// TIA Portal project "Projecto3Automação_1500_V18" (V18)

(* hardware
DEVICE "S71500/ET200MP station_1"  S7-1500 station
   slot 0: "Rail_0"  Rack  6ES7 590-1***0-0AA0
   slot 0: "PM 190W 120/230VAC"  PM 190W 120/230VAC  6EP1333-4BA00
   slot 1: "PLC_1"  CPU 1516-3 PN/DP  6ES7 516-3AN02-0AB0  V2.8
      slot 3: "CPU display_1"  6ES7591-1BA00-0AA0
      slot 32768: "PROFINET interface_1"  X1
         slot 32769: "Port_1"  X1 P1
         slot 32770: "Port_2"  X1 P2
      slot 33024: "PROFINET interface_2"  X2
         slot 33025: "Port_1"  X2 P1
      slot 33280: "DP interface_1"  X3
      slot 34817: "Virtual CP interface port_1"  Virtual CP interface port  Virtual CP interface port
   slot 2: "DI 32x24VDC HF_1"  DI 32x24VDC HF  6ES7 521-1BL00-0AB0  V2.2
   slot 3: "DQ 32x24VDC/0.5A HF_1"  DQ 32x24VDC/0.5A HF  6ES7 522-1BL01-0AB0  V1.1
   slot 4: "AI 8xU/I/RTD/TC ST_1"  AI 8xU/I/RTD/TC ST  6ES7 531-7KF00-0AB0  V2.2
   slot 5: "AQ 4xU/I ST_1"  AQ 4xU/I ST  6ES7 532-5HD00-0AB0  V2.2
DEVICE "PC station"  SIMATIC PC station
   slot 0: "PC station"  Rail  SIMATIC PC-Station  V1.0
      slot 125: "Stationmanager"  Station_Manager  V6.0.4
   slot 1: "HMI_RT_1"  WinCC RT Advanced  6AV2 104-0xxxx-xxxx  16.0.0.0
      slot 33792: "Computer interface"  Host interface
   slot 2: "IE general_1"  IE General  IE_CP  V8.2.0
DEVICE "S7-1500/ET200MP station_1"  S7-1500 station
   slot 0: "Rail_0"  Rack  6ES7 590-1***0-0AA0
   slot 1: "PLC_2"  CPU 1512C-1 PN  6ES7 512-1CK01-0AB0  V2.9
      slot 3: "CPU display_1"  6ES7591-1AA00-0AA0
      slot 32768: "PROFINET interface_1"  X1
         slot 32769: "Port_1"  X1 P1
         slot 32770: "Port_2"  X1 P2
      slot 34817: "Virtual CP interface port_1"  Virtual CP interface port  Virtual CP interface port
*)

// ===== PLC "PLC_1"  CPU 1516-3 PN/DP =====

VAR_GLOBAL   // PLC tag table "Default tag table"
   "Sensor Tapete 1 Entrada 1" AT %I10.0 : Bool;
   "Sensor Tapete 2 Entrada 2" AT %I10.1 : Bool;
   "Sensor Inicial Tapete 3 Saida 1" AT %I10.2 : Bool;
   "Sensor Final Tapete 3 Saida 1" AT %I10.3 : Bool;
   "Sensor Inicial Tapete 4 Saida 2" AT %I10.4 : Bool;
   "Sensor Final Tapete 4 Saida 2" AT %I10.5 : Bool;
   "Sensor Final Tapete 6 Saida 2" AT %I10.6 : Bool;
   "Sensor Final Tapete 7" AT %I10.7 : Bool;
   "Sensor  Grampo Aperto" AT %I11.0 : Bool;
   "Sensor Posicionador Cima/Baixo" AT %I11.1 : Bool;
   "Sensor Posicionador Frente/Tras" AT %I11.2 : Bool;
   "Sensor Posicionador Presença Peça" AT %I11.3 : Bool;
   "Sensor Saida Posto 1" AT %I11.4 : Bool;
   "Sensor Saida Posto 2" AT %I11.5 : Bool;
   "Sensor Saida Posto 3" AT %I11.6 : Bool;
   "Sensor Saida Posto 4" AT %I11.7 : Bool;
   "Sensor Saida Posto 5" AT %I12.0 : Bool;
   "Sensor Saida Posto 6" AT %I12.1 : Bool;
   "Emissor 1" AT %Q10.0 : Bool;
   "Tapete 1" AT %Q10.1 : Bool;
   "C. Maq. 1 Ativa" AT %Q10.2 : Bool;
   "C. Maq. 1 Parar" AT %Q10.3 : Bool;
   "C. Maq. 1 Bases/Tampas" AT %Q10.4 : Bool;
   "Emissor 2" AT %Q10.5 : Bool;
   "Tapete 2" AT %Q10.6 : Bool;
   "C. Maq. 2 Ativa" AT %Q10.7 : Bool;
   "C. Maq. 2 Parar" AT %Q11.0 : Bool;
   "C. Maq. 2 Bases/Tampas" AT %Q11.1 : Bool;
   "Grampo Aperto" AT %Q11.2 : Bool;
   "Grampo Levantar" AT %Q11.3 : Bool;
   "Posicionador Cima/Baixo" AT %Q11.4 : Bool;
   "Posicionador Frente/Tras" AT %Q11.5 : Bool;
   "Posicionador Vacuo" AT %Q11.6 : Bool;
   "Direcionador 1 Ligar" AT %Q12.0 : Bool;
   "Direcionador 1 Direita" AT %Q12.1 : Bool;
   "Direcionador 1 Esquerda" AT %Q12.2 : Bool;
   "Direcionador 2 Ligar" AT %Q12.3 : Bool;
   "Direcionador 2 Direita" AT %Q12.4 : Bool;
   "Direcionador 2 Esquerda" AT %Q12.5 : Bool;
   "Barreira Posto 3 e 5" AT %Q12.6 : Bool;
   "Barreira Posto 2 e 4" AT %Q12.7 : Bool;
   "C. Maq. 1 em Processo" AT %ID100 : DInt;
   "C. Maq. 2 em Processo" AT %ID104 : DInt;
   "Tapete 3" AT %QD100 : Real;
   "Tapete 4" AT %QD104 : Real;
   "Tapete 5" AT %QD108 : Real;
   "Tapete 6" AT %QD112 : Real;
   "Valvula Enchimento Tanque 1" AT %QD120 : Real;   // analog output manipulated value pump1
   "Valvula Descarga Tanque 1" AT %QD124 : Real;
   "Valvula Enchimento Tanque 2" AT %QD128 : Real;   // analog output manipulated value pump2
   "Valvula Descarga Tanque 2" AT %QD132 : Real;
   "Contador 1" AT %QD136 : DInt;
   "Contador 2" AT %QD140 : DInt;
   "Ordem de arranque" AT %M100.0 : Bool;
   "Ordem de paragem" AT %M100.1 : Bool;
   "M_Tapete1" AT %M103.0 : Bool;
   "M_Tapete2" AT %M103.1 : Bool;
   "M_Tapete3" AT %M103.2 : Bool;
   "M_Tapete4" AT %M103.3 : Bool;
   "M_Tapete5" AT %M103.4 : Bool;
   "M_Tapete6" AT %M103.5 : Bool;
   "M_Tapete7" AT %M103.6 : Bool;
   "V_Tapete3" AT %MD300 : Real;
   "V_Tapete4" AT %MD400 : Real;
   "V_Tapete5" AT %MD500 : Real;
   "V_Tapete6" AT %MD600 : Real;
   "V_Tapete7" AT %MD700 : Real;
   "Etapa_0" AT %M102.7 : Bool;
   "Etapa_1" AT %M103.7 : Bool;
   "Etapa_2" AT %M104.0 : Bool;
   "Etapa_3" AT %M104.1 : Bool;
   "Etapa_4" AT %M104.2 : Bool;
   "Etapa_5" AT %M104.3 : Bool;
   "Etapa_6" AT %M104.4 : Bool;
   "Etapa_7" AT %M104.5 : Bool;
   "Etapa_8" AT %M104.6 : Bool;
   "Etapa_9" AT %M104.7 : Bool;
   "Etapa_10" AT %M105.0 : Bool;
   "Etapa_11" AT %M105.1 : Bool;
   "Etapa_30" AT %M105.2 : Bool;
   "Etapa_31" AT %M105.3 : Bool;
   "Etapa_32" AT %M105.4 : Bool;
   "Etapa_33" AT %M105.5 : Bool;
   "Etapa_34" AT %M105.6 : Bool;
   "NPosto" AT %MW1000 : Int;
   "Etapa_12" AT %M105.7 : Bool;
   "Etapa_13" AT %M106.0 : Bool;
   "Etapa_14" AT %M106.1 : Bool;
   "Etapa_15" AT %M106.2 : Bool;
   "Etapa_20" AT %M106.3 : Bool;
   "Etapa_35" AT %M106.4 : Bool;
   "Etapa_36" AT %M106.5 : Bool;
   "Etapa_37" AT %M106.6 : Bool;
   "Etapa_38" AT %M106.7 : Bool;
   "Etapa_39" AT %M107.0 : Bool;
   "Etapa_40" AT %M107.1 : Bool;
   "Etapa_50" AT %M107.2 : Bool;
   "Empilhar" AT %M70.0 : Bool;
   "Sensor_Geral_Posto" AT %M170.0 : Bool;
   "Fim de ciclo" AT %M107.5 : Bool;
   "Sensor Grampo Levantar" AT %I12.2 : Bool;
   "Entrada_Base" AT %M107.6 : Bool;
   "Move Nposto 1" AT %M170.1 : Bool;
   "Etapa_100" AT %M150.0 : Bool;
   "Etapa_101" AT %M150.1 : Bool;
   "Etapa_102" AT %M150.2 : Bool;
   "Etapa_103" AT %M150.3 : Bool;
   "Etapa_104" AT %M150.4 : Bool;
   "Etapa_105" AT %M150.5 : Bool;
   "Etapa_106" AT %M150.6 : Bool;
   "Etapa_107" AT %M150.7 : Bool;
   "Etapa_110" AT %M151.0 : Bool;
   "Etapa_111" AT %M151.1 : Bool;
   "Etapa_112" AT %M151.2 : Bool;
   "Etapa_113" AT %M151.3 : Bool;
   "Etapa_114" AT %M151.4 : Bool;
   "Etapa_115" AT %M151.5 : Bool;
   "Etapa_116" AT %M151.6 : Bool;
   "Etapa_117" AT %M151.7 : Bool;
   "Etapa_120" AT %M152.0 : Bool;
   "Etapa_121" AT %M152.1 : Bool;
   "Etapa_122" AT %M152.2 : Bool;
   "Etapa_123" AT %M152.3 : Bool;
   "Etapa_124" AT %M152.4 : Bool;
   "Etapa_125" AT %M152.5 : Bool;
   "Etapa_126" AT %M152.6 : Bool;
   "Etapa_127" AT %M152.7 : Bool;
   "Etapa_130" AT %M153.0 : Bool;
   "Etapa_131" AT %M153.1 : Bool;
   "Etapa_132" AT %M153.2 : Bool;
   "Etapa_133" AT %M153.3 : Bool;
   "Etapa_134" AT %M153.4 : Bool;
   "Etapa_135" AT %M153.5 : Bool;
   "Etapa_136" AT %M153.6 : Bool;
   "Etapa_137" AT %M153.7 : Bool;
   "Etapa_150" AT %M155.0 : Bool;
   "Etapa_151" AT %M155.1 : Bool;
   "Etapa_152" AT %M155.2 : Bool;
   "Etapa_153" AT %M155.3 : Bool;
   "Etapa_154" AT %M155.4 : Bool;
   "Etapa_155" AT %M155.5 : Bool;
   "Etapa_156" AT %M155.6 : Bool;
   "Etapa_157" AT %M155.7 : Bool;
   "Pedido_Posic_Ao_Tapete_3" AT %M160.0 : Bool;
   "Pedido_Posic_Ao_Tapete_6" AT %M160.1 : Bool;
   "Pedido_Tap6_Ao_Tapete_4" AT %M160.2 : Bool;
   "Habilita_Remover_1" AT %M61.0 : Bool;
   "Habilita_Remover_2" AT %M61.1 : Bool;
   "Habilita_Remover_3" AT %M61.2 : Bool;
   "Habilita_Remover_4" AT %M61.3 : Bool;
   "Habilita_Remover_5" AT %M61.4 : Bool;
   "Habilita_Remover_6" AT %M61.5 : Bool;
   "Habilita_Máquina_1" AT %M61.6 : Bool;
   "Habilita_Máquina_2" AT %M61.7 : Bool;
   "Máquina1_Tampas" AT %M62.0 : Bool;
   "Máquina2_Tampas" AT %M62.1 : Bool;
   "Etapa_16" AT %M107.4 : Bool;
   "Scan_Estado_31" AT %M165.0 : Bool;
   "Contador_Remover_1" AT %MD10 : DWord;
   "Contador_Remover_2" AT %MD14 : DWord;
   "Contador_Remover_3" AT %MD18 : DWord;
   "Contador_Remover_4" AT %MD22 : DWord;
   "Contador_Remover_5" AT %MD26 : DWord;
   "Contador_Remover_6" AT %MD30 : DWord;
   "Start" AT %M100.2 : Bool;
   "Stop" AT %M100.3 : Bool;
   "Emergência" AT %M180.0 : Bool;
   "Reset" AT %M100.5 : Bool;
   "Nivel_Tanque_1" AT %ID108 : Real;   // analog Input actual level filing level Tank1
   "Nivel_Tanque_2" AT %ID112 : Real;   // analog Input actual level filing level Tank2
   "S1" AT %I150.0 : Bool;   // sudden setpoint change filing level 0 (0) or 700 (1)
   "Tapete 7" AT %QD116 : Real;
   "Algum_Remover_Habilitado" AT %M100.6 : Bool;
   "Algum_Máquina_Habilitada" AT %M100.7 : Bool;
   "Sem_Condições_Empilhar" AT %M101.0 : Bool;
   "Primeiro_Scan" AT %M200.0 : Bool;
   "Aviso_Sem_Condições_Empilhar" AT %M154.0 : Bool;
   "Aviso_Nenhuma_Máquina_Habilitada" AT %M158.0 : Bool;
   "Aviso_Nenhum_Remover_Habilitado" AT %M162.0 : Bool;
   "Contador_Remover_Total" AT %MD34 : DWord;
   "Aviso_Sem_Condições_Empilhar(1)" AT %MW154 : Int;
   "Aviso_Nenhuma_Máquina_Habilitada(1)" AT %MW158 : Int;
   "Aviso_Nenhum_Remover_Habilitado(1)" AT %MW162 : Int;
   "Contador_Máquina_1" AT %MD38 : DWord;
   "Contador_Máquina_2" AT %MD42 : DWord;
   "Nivel_1_convertido" AT %MD50 : Real;
   "Nivel_1_convertido_Scada" AT %ID60 : Real;
   "Reset Contadores Postos" AT %M700.0 : Bool;
   "Reset Contadores Maquinas" AT %M704.0 : Bool;
   "Nivel_2_convertido" AT %MD54 : Real;
   "Nivel_2_convertido_Scada" AT %ID64 : Real;
   "Emergencia Scada" AT %MW166 : Int;
   "Ret_value" AT %MW168 : Int;
   "Reset_Cont_Diario" AT %MD46 : DWord;
   "Tag_1" AT %MD174 : DWord;
   "Ordem de arranque s ordem paragem" AT %M100.4 : Bool;
   "Contador_Remover_1_Anterior" AT %MD310 : DWord;
   "Contador_Remover_2_Anterior" AT %MD314 : DWord;
   "Contador_Remover_3_Anterior" AT %MD318 : DWord;
   "Contador_Remover_4_Anterior" AT %MD322 : DWord;
   "Contador_Remover_5_Anterior" AT %MD326 : DWord;
   "Contador_Remover_6_Anterior" AT %MD330 : DWord;
   "Contador_Máquina_1_Anterior" AT %MD334 : DWord;
   "Contador_Máquina_2_Anterior" AT %MD338 : DWord;
   "Trigger_Contador" AT %M342.0 : Bool;
   "Set_vel_T3" AT %MD342 : Real;
   "Set_vel_T4" AT %MD346 : Real;
   "Set_vel_T5" AT %MD350 : Real;
   "Set_vel_T6" AT %MD354 : Real;
   "Set_vel_T7" AT %MD358 : Real;
   "Clock_1Hz" AT %M1100.5 : Bool;
   "Clock_2.5Hz" AT %M1100.2 : Bool;
   "Clock_2Hz" AT %M1100.3 : Bool;
END_VAR

DATA_BLOCK "Pulse"   // DB1
{ S7_Optimized_Access := 'TRUE' }
VERSION : 0.1
   VAR
      Pulse1 : Bool;
      Pulse2 : Bool;
      Pulse3 : Bool;
      Pulse4 : Bool;
      Pulse5 : Bool;
      Pulse6 : Bool;
      Pulse7 : Bool;
      Pulse8 : Bool;
      Pulse9 : Bool;
      Pulse10 : Bool;
      Pulse11 : Bool;
      Pulse12 : Bool;
      Pulse13 : Bool;
      Pulse14 : Bool;
      Pulse15 : Bool;
      Pulse16 : Bool;
      Pulse17 : Bool;
      Pulse18 : Bool;
      Pulse19 : Bool;
      Pulse20 : Bool;
      Pulse21 : Bool;
      Pulse22 : Bool;
      Pulse23 : Bool;
      Pulse24 : Bool;
      pulse25 : Bool;
      pulse26 : Bool;
      pulse27 : Bool;
      pulse28 : Bool;
      pulse29 : Bool;
      pulse30 : Bool;
      pulse31 : Bool;
      pulse32 : Bool;
      pulse33 : Bool;
   END_VAR
BEGIN
END_DATA_BLOCK

DATA_BLOCK "PLC1_Data_Sent"   // DB19
{ S7_Optimized_Access := 'FALSE' }
VERSION : 0.1
   VAR
      Contador_Remover_1 : DWord;
      Contador_Remover_2 : DWord;
      Contador_Remover_3 : DWord;
      Contador_Remover_4 : DWord;
      Contador_Remover_5 : DWord;
      Contador_Remover_6 : DWord;
      Contador_Remover_Total : DWord;
      Contador_Máquina_1 : DWord;
      Contador_Máquina_2 : DWord;
      "Valvula Enchimento Tanque 1" : Real;
      "Valvula Descarga Tanque 1" : Real;
      "Valvula Enchimento Tanque 2" : Real;
      "Valvula Descarga Tanque 2" : Real;
      Nivel_1_convertido_Scada : Real;
      Nivel_2_convertido_Scada : Real;
      Aviso_Nenhuma_Máquina_Habilitada : Bool;
      Aviso_Nenhum_Remover_Habilitado : Bool;
      Aviso_Sem_Condições_Empilhar : Bool;
      OUT_Set_vel_T3 : Real;
      OUT_Set_vel_T4 : Real;
      OUT_Set_vel_T5 : Real;
      OUT_Set_vel_T6 : Real;
      OUT_Set_vel_T7 : Real;
   END_VAR
BEGIN
END_DATA_BLOCK

DATA_BLOCK "PLC1_Data_Received"   // DB22
{ S7_Optimized_Access := 'FALSE' }
VERSION : 0.1
   VAR
      Start : Bool;
      Stop : Bool;
      Emergência : Bool;
      Habilita_Remover_1 : Bool;
      Habilita_Remover_2 : Bool;
      Habilita_Remover_3 : Bool;
      Habilita_Remover_4 : Bool;
      Habilita_Remover_5 : Bool;
      Habilita_Remover_6 : Bool;
      Habilita_Máquina_1 : Bool;
      Habilita_Máquina_2 : Bool;
      Empilhar : Bool;
      Reset_Cont_Diario : DWord;
      "Reset Contadores Maquinas" : Bool;
      "Reset Contadores Postos" : Bool;
      Máquina2_Tampas : Bool;
      Máquina1_Tampas : Bool;
   END_VAR
BEGIN
END_DATA_BLOCK

// folder: System blocks/Program resources

DATA_BLOCK "TempVacuo1"   // DB2
{ S7_Optimized_Access := 'TRUE' }
AUTHOR : Simatic
FAMILY : IEC
NAME : IEC_TMR
VERSION : 1.0
// stored: InstanceOfName IEC_TIMER
"IEC_TIMER"
BEGIN
END_DATA_BLOCK

DATA_BLOCK "TempVacuo2"   // DB3
{ S7_Optimized_Access := 'TRUE' }
AUTHOR : Simatic
FAMILY : IEC
NAME : IEC_TMR
VERSION : 1.0
// stored: InstanceOfName IEC_TIMER
"IEC_TIMER"
BEGIN
END_DATA_BLOCK

DATA_BLOCK "Temporizador_Aviso_Remover"   // DB4
{ S7_Optimized_Access := 'TRUE' }
AUTHOR : Simatic
FAMILY : IEC
NAME : IEC_TMR
VERSION : 1.0
// stored: InstanceOfName IEC_TIMER
"IEC_TIMER"
BEGIN
END_DATA_BLOCK

DATA_BLOCK "Temporizador_Aviso_Máquina"   // DB5
{ S7_Optimized_Access := 'TRUE' }
AUTHOR : Simatic
FAMILY : IEC
NAME : IEC_TMR
VERSION : 1.0
// stored: InstanceOfName IEC_TIMER
"IEC_TIMER"
BEGIN
END_DATA_BLOCK

DATA_BLOCK "Temp_300ms_T3"   // DB6
{ S7_Optimized_Access := 'TRUE' }
AUTHOR : Simatic
FAMILY : IEC
NAME : IEC_TMR
VERSION : 1.0
// stored: InstanceOfName IEC_TIMER
"IEC_TIMER"
BEGIN
END_DATA_BLOCK

DATA_BLOCK "T300ms"   // DB7
{ S7_Optimized_Access := 'TRUE' }
AUTHOR : Simatic
FAMILY : IEC
NAME : IEC_TMR
VERSION : 1.0
// stored: InstanceOfName IEC_TIMER
"IEC_TIMER"
BEGIN
END_DATA_BLOCK

DATA_BLOCK "Temp_300ms_T4"   // DB8
{ S7_Optimized_Access := 'TRUE' }
AUTHOR : Simatic
FAMILY : IEC
NAME : IEC_TMR
VERSION : 1.0
// stored: InstanceOfName IEC_TIMER
"IEC_TIMER"
BEGIN
END_DATA_BLOCK

DATA_BLOCK "Temporizador_Aviso_Empilhar"   // DB13
{ S7_Optimized_Access := 'TRUE' }
AUTHOR : Simatic
FAMILY : IEC
NAME : IEC_TMR
VERSION : 1.0
// stored: InstanceOfName IEC_TIMER
"IEC_TIMER"
BEGIN
END_DATA_BLOCK

DATA_BLOCK "Tempo"   // DB14
{ S7_Optimized_Access := 'TRUE' }
VERSION : 0.1
   VAR
      Tempo_dia : DTL;
   END_VAR
BEGIN
END_DATA_BLOCK

DATA_BLOCK "Temp_100ms"   // DB15
{ S7_Optimized_Access := 'TRUE' }
AUTHOR : Simatic
FAMILY : IEC
NAME : IEC_TMR
VERSION : 1.0
// stored: InstanceOfName IEC_TIMER
"IEC_TIMER"
BEGIN
END_DATA_BLOCK

DATA_BLOCK "Temp_3s"   // DB17
{ S7_Optimized_Access := 'TRUE' }
AUTHOR : Simatic
FAMILY : IEC
NAME : IEC_TMR
VERSION : 1.0
// stored: InstanceOfName IEC_TIMER
"IEC_TIMER"
BEGIN
END_DATA_BLOCK

DATA_BLOCK "PLC_1_Send_DB"   // DB18
{ S7_Optimized_Access := 'TRUE' }
AUTHOR : SIMATIC
FAMILY : MC7Plus
NAME : TC_IP_v4
VERSION : 1.0
// stored: InstanceOfName TCON_IP_v4
"TCON_IP_v4"
BEGIN
   ID := 1;
   InterfaceId := 64;
   RemotePort := 2000;
   ActiveEstablished := true;
   RemoteAddress.ADDR[1] := 192;
   RemoteAddress.ADDR[2] := 168;
   RemoteAddress.ADDR[3] := 228;
   RemoteAddress.ADDR[4] := 55;
END_DATA_BLOCK

DATA_BLOCK "PLC_1_Receive_DB"   // DB21
{ S7_Optimized_Access := 'TRUE' }
AUTHOR : SIMATIC
FAMILY : MC7Plus
NAME : TC_IP_v4
VERSION : 1.0
// stored: InstanceOfName TCON_IP_v4
"TCON_IP_v4"
BEGIN
   ID := 2;
   InterfaceId := 64;
   LocalPort := 2000;
   RemoteAddress.ADDR[1] := 192;
   RemoteAddress.ADDR[2] := 168;
   RemoteAddress.ADDR[3] := 228;
   RemoteAddress.ADDR[4] := 55;
END_DATA_BLOCK

// folder: (top level)

FUNCTION "Centro Maquinação 1" : Void   // FC1, LAD
TITLE = Centro de Maquinação 1
{ S7_Optimized_Access := 'TRUE' }
VERSION : 0.1
   VAR_TEMP   // added for the SCL form of the ladder/FBD networks
      _w1 : Bool;
   END_VAR
BEGIN

REGION Network 1: Peça nova para entrada na máquina 1
   // Quando a peça atravessa o sensor do tapete 1 podemos ligar a máquina 1 para a recolher
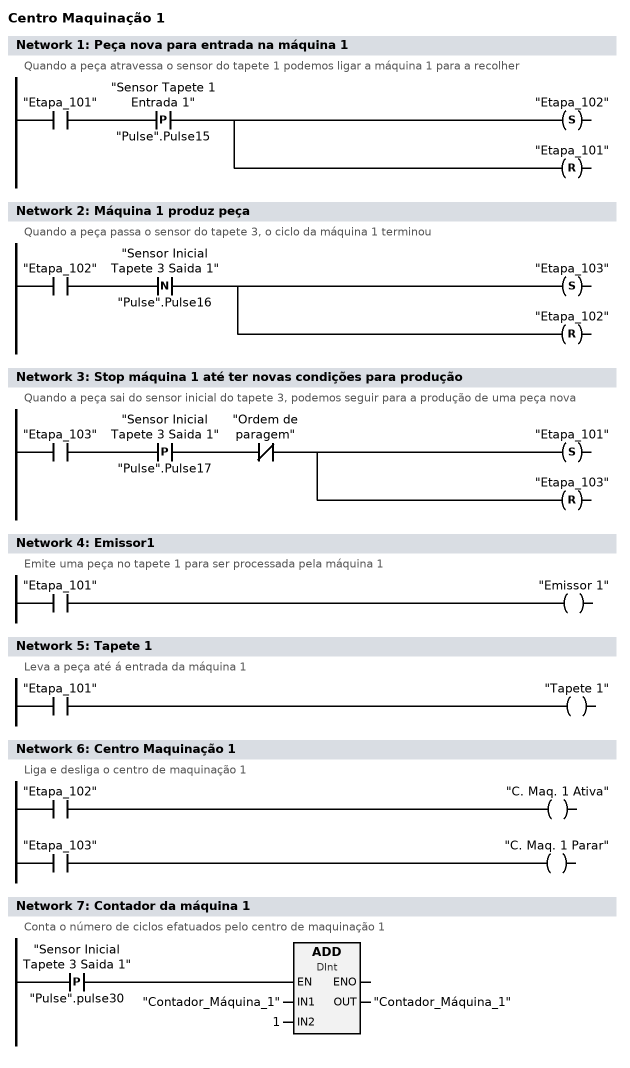
   RUNG wire#powerrail
      Contact( "Etapa_101" )
      P_Contact(operand := "Sensor Tapete 1 Entrada 1", bit := "Pulse".Pulse15)
      wire#w1
      S_Coil( "Etapa_102" )
   END_RUNG
   RUNG wire#w1
      R_Coil( "Etapa_101" )
   END_RUNG
   // the same network as SCL:
   #_w1 := "Etapa_101" AND "Sensor Tapete 1 Entrada 1" AND NOT "Pulse".Pulse15;   // rising edge of "Sensor Tapete 1 Entrada 1"
   "Pulse".Pulse15 := "Sensor Tapete 1 Entrada 1";
   IF #_w1 THEN
       "Etapa_102" := TRUE;
       "Etapa_101" := FALSE;
   END_IF;
END_REGION

REGION Network 2: Máquina 1 produz peça
   // Quando a peça passa o sensor do tapete 3, o ciclo da máquina 1 terminou
   RUNG wire#powerrail
      Contact( "Etapa_102" )
      N_Contact(operand := "Sensor Inicial Tapete 3 Saida 1", bit := "Pulse".Pulse16)
      wire#w1
      S_Coil( "Etapa_103" )
   END_RUNG
   RUNG wire#w1
      R_Coil( "Etapa_102" )
   END_RUNG
   // the same network as SCL:
   #_w1 := "Etapa_102" AND NOT "Sensor Inicial Tapete 3 Saida 1" AND "Pulse".Pulse16;   // falling edge of "Sensor Inicial Tapete 3 Saida 1"
   "Pulse".Pulse16 := "Sensor Inicial Tapete 3 Saida 1";
   IF #_w1 THEN
       "Etapa_103" := TRUE;
       "Etapa_102" := FALSE;
   END_IF;
END_REGION

REGION Network 3: Stop máquina 1 até ter novas condições para produção
   // Quando a peça sai do sensor inicial do tapete 3, podemos seguir para a produção de uma peça nova
   RUNG wire#powerrail
      Contact( "Etapa_103" )
      P_Contact(operand := "Sensor Inicial Tapete 3 Saida 1", bit := "Pulse".Pulse17)
      I_Contact( "Ordem de paragem" )
      wire#w1
      S_Coil( "Etapa_101" )
   END_RUNG
   RUNG wire#w1
      R_Coil( "Etapa_103" )
   END_RUNG
   // the same network as SCL:
   #_w1 := "Etapa_103" AND "Sensor Inicial Tapete 3 Saida 1" AND NOT "Pulse".Pulse17;   // rising edge of "Sensor Inicial Tapete 3 Saida 1"
   "Pulse".Pulse17 := "Sensor Inicial Tapete 3 Saida 1";
   IF #_w1 AND NOT "Ordem de paragem" THEN
       "Etapa_101" := TRUE;
       "Etapa_103" := FALSE;
   END_IF;
END_REGION

REGION Network 4: Emissor1
   // Emite uma peça no tapete 1 para ser processada pela máquina 1
   RUNG wire#powerrail
      Contact( "Etapa_101" )
      Coil( "Emissor 1" )
   END_RUNG
   // the same network as SCL:
   "Emissor 1" := "Etapa_101";
END_REGION

REGION Network 5: Tapete 1
   // Leva a peça até á entrada da máquina 1
   RUNG wire#powerrail
      Contact( "Etapa_101" )
      Coil( "Tapete 1" )
   END_RUNG
   // the same network as SCL:
   "Tapete 1" := "Etapa_101";
END_REGION

REGION Network 6: Centro Maquinação 1
   // Liga e desliga o centro de maquinação 1
   RUNG wire#powerrail
      Contact( "Etapa_102" )
      Coil( "C. Maq. 1 Ativa" )
   END_RUNG
   RUNG wire#powerrail
      Contact( "Etapa_103" )
      Coil( "C. Maq. 1 Parar" )
   END_RUNG
   // the same network as SCL:
   "C. Maq. 1 Ativa" := "Etapa_102";
   "C. Maq. 1 Parar" := "Etapa_103";
END_REGION

REGION Network 7: Contador da máquina 1
   // Conta o número de ciclos efatuados pelo centro de maquinação 1
   RUNG wire#powerrail
      P_Contact(operand := "Sensor Inicial Tapete 3 Saida 1", bit := "Pulse".pulse30)
      { S7_Templates := "SrcType := DInt" } Add(in1 := "Contador_Máquina_1", in2 := 1, out => "Contador_Máquina_1")
   END_RUNG
   // the same network as SCL:
   #_w1 := "Sensor Inicial Tapete 3 Saida 1" AND NOT "Pulse".pulse30;   // rising edge of "Sensor Inicial Tapete 3 Saida 1"
   "Pulse".pulse30 := "Sensor Inicial Tapete 3 Saida 1";
   IF #_w1 THEN "Contador_Máquina_1" := "Contador_Máquina_1" + 1; END_IF;
END_REGION
END_FUNCTION

FUNCTION "Centro Maquinação 2" : Void   // FC2, LAD
TITLE = Centro de Maquinação 2
{ S7_Optimized_Access := 'TRUE' }
VERSION : 0.1
   VAR_TEMP   // added for the SCL form of the ladder/FBD networks
      _w1 : Bool;
   END_VAR
BEGIN

REGION Network 1: Peça nova para entrada na máquina 2
   // Quando a peça atravessa o sensor do tapete 2 podemos ligar a máquina 2 para a recolher
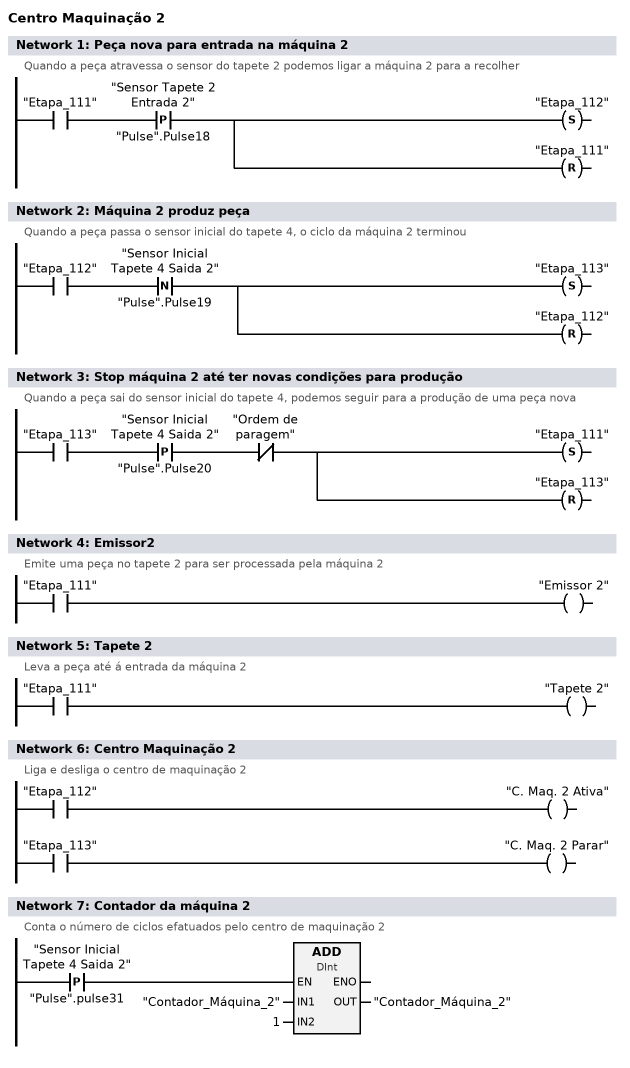
   RUNG wire#powerrail
      Contact( "Etapa_111" )
      P_Contact(operand := "Sensor Tapete 2 Entrada 2", bit := "Pulse".Pulse18)
      wire#w1
      S_Coil( "Etapa_112" )
   END_RUNG
   RUNG wire#w1
      R_Coil( "Etapa_111" )
   END_RUNG
   // the same network as SCL:
   #_w1 := "Etapa_111" AND "Sensor Tapete 2 Entrada 2" AND NOT "Pulse".Pulse18;   // rising edge of "Sensor Tapete 2 Entrada 2"
   "Pulse".Pulse18 := "Sensor Tapete 2 Entrada 2";
   IF #_w1 THEN
       "Etapa_112" := TRUE;
       "Etapa_111" := FALSE;
   END_IF;
END_REGION

REGION Network 2: Máquina 2 produz peça
   // Quando a peça passa o sensor inicial do tapete 4, o ciclo da máquina 2 terminou
   RUNG wire#powerrail
      Contact( "Etapa_112" )
      N_Contact(operand := "Sensor Inicial Tapete 4 Saida 2", bit := "Pulse".Pulse19)
      wire#w1
      S_Coil( "Etapa_113" )
   END_RUNG
   RUNG wire#w1
      R_Coil( "Etapa_112" )
   END_RUNG
   // the same network as SCL:
   #_w1 := "Etapa_112" AND NOT "Sensor Inicial Tapete 4 Saida 2" AND "Pulse".Pulse19;   // falling edge of "Sensor Inicial Tapete 4 Saida 2"
   "Pulse".Pulse19 := "Sensor Inicial Tapete 4 Saida 2";
   IF #_w1 THEN
       "Etapa_113" := TRUE;
       "Etapa_112" := FALSE;
   END_IF;
END_REGION

REGION Network 3: Stop máquina 2 até ter novas condições para produção
   // Quando a peça sai do sensor inicial do tapete 4, podemos seguir para a produção de uma peça nova
   RUNG wire#powerrail
      Contact( "Etapa_113" )
      P_Contact(operand := "Sensor Inicial Tapete 4 Saida 2", bit := "Pulse".Pulse20)
      I_Contact( "Ordem de paragem" )
      wire#w1
      S_Coil( "Etapa_111" )
   END_RUNG
   RUNG wire#w1
      R_Coil( "Etapa_113" )
   END_RUNG
   // the same network as SCL:
   #_w1 := "Etapa_113" AND "Sensor Inicial Tapete 4 Saida 2" AND NOT "Pulse".Pulse20;   // rising edge of "Sensor Inicial Tapete 4 Saida 2"
   "Pulse".Pulse20 := "Sensor Inicial Tapete 4 Saida 2";
   IF #_w1 AND NOT "Ordem de paragem" THEN
       "Etapa_111" := TRUE;
       "Etapa_113" := FALSE;
   END_IF;
END_REGION

REGION Network 4: Emissor2
   // Emite uma peça no tapete 2 para ser processada pela máquina 2
   RUNG wire#powerrail
      Contact( "Etapa_111" )
      Coil( "Emissor 2" )
   END_RUNG
   // the same network as SCL:
   "Emissor 2" := "Etapa_111";
END_REGION

REGION Network 5: Tapete 2
   // Leva a peça até á entrada da máquina 2
   RUNG wire#powerrail
      Contact( "Etapa_111" )
      Coil( "Tapete 2" )
   END_RUNG
   // the same network as SCL:
   "Tapete 2" := "Etapa_111";
END_REGION

REGION Network 6: Centro Maquinação 2
   // Liga e desliga o centro de maquinação 2
   RUNG wire#powerrail
      Contact( "Etapa_112" )
      Coil( "C. Maq. 2 Ativa" )
   END_RUNG
   RUNG wire#powerrail
      Contact( "Etapa_113" )
      Coil( "C. Maq. 2 Parar" )
   END_RUNG
   // the same network as SCL:
   "C. Maq. 2 Ativa" := "Etapa_112";
   "C. Maq. 2 Parar" := "Etapa_113";
END_REGION

REGION Network 7: Contador da máquina 2
   // Conta o número de ciclos efatuados pelo centro de maquinação 2
   RUNG wire#powerrail
      P_Contact(operand := "Sensor Inicial Tapete 4 Saida 2", bit := "Pulse".pulse31)
      { S7_Templates := "SrcType := DInt" } Add(in1 := "Contador_Máquina_2", in2 := 1, out => "Contador_Máquina_2")
   END_RUNG
   // the same network as SCL:
   #_w1 := "Sensor Inicial Tapete 4 Saida 2" AND NOT "Pulse".pulse31;   // rising edge of "Sensor Inicial Tapete 4 Saida 2"
   "Pulse".pulse31 := "Sensor Inicial Tapete 4 Saida 2";
   IF #_w1 THEN "Contador_Máquina_2" := "Contador_Máquina_2" + 1; END_IF;
END_REGION
END_FUNCTION

FUNCTION "Conversões" : Void   // FC3, LAD
TITLE = Conversões
{ S7_Optimized_Access := 'TRUE' }
VERSION : 0.1
   VAR_TEMP
      Erro : Int;
      aux1 : Int;
   END_VAR
BEGIN

REGION Network 1: Conversão Tapete3
   // Conversão para ajuste da velocidade do tapete 3
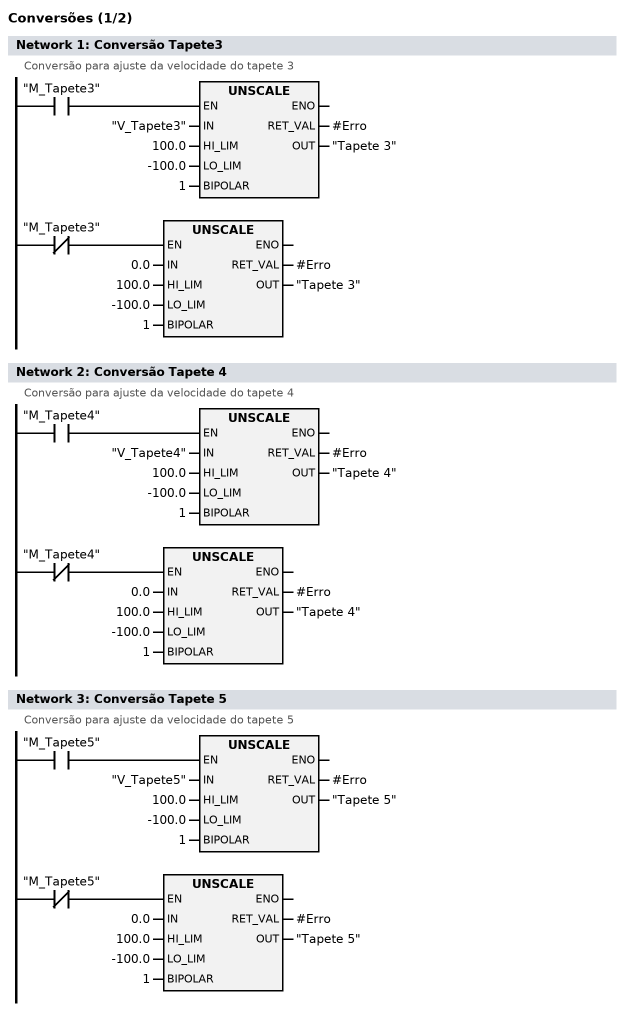
   IF "M_Tapete3" THEN
       #Erro := UNSCALE(IN := "V_Tapete3", HI_LIM := 100.0, LO_LIM := -100.0, BIPOLAR := 1, OUT => "Tapete 3");
   END_IF;
   IF NOT "M_Tapete3" THEN
       #Erro := UNSCALE(IN := 0.0, HI_LIM := 100.0, LO_LIM := -100.0, BIPOLAR := 1, OUT => "Tapete 3");
   END_IF;
END_REGION

REGION Network 2: Conversão Tapete 4
   // Conversão para ajuste da velocidade do tapete 4
   IF "M_Tapete4" THEN
       #Erro := UNSCALE(IN := "V_Tapete4", HI_LIM := 100.0, LO_LIM := -100.0, BIPOLAR := 1, OUT => "Tapete 4");
   END_IF;
   IF NOT "M_Tapete4" THEN
       #Erro := UNSCALE(IN := 0.0, HI_LIM := 100.0, LO_LIM := -100.0, BIPOLAR := 1, OUT => "Tapete 4");
   END_IF;
END_REGION

REGION Network 3: Conversão Tapete 5
   // Conversão para ajuste da velocidade do tapete 5
   IF "M_Tapete5" THEN
       #Erro := UNSCALE(IN := "V_Tapete5", HI_LIM := 100.0, LO_LIM := -100.0, BIPOLAR := 1, OUT => "Tapete 5");
   END_IF;
   IF NOT "M_Tapete5" THEN
       #Erro := UNSCALE(IN := 0.0, HI_LIM := 100.0, LO_LIM := -100.0, BIPOLAR := 1, OUT => "Tapete 5");
   END_IF;
END_REGION

REGION Network 4: Conversão Tapete 6
   // Conversão para ajuste da velocidade do tapete 6
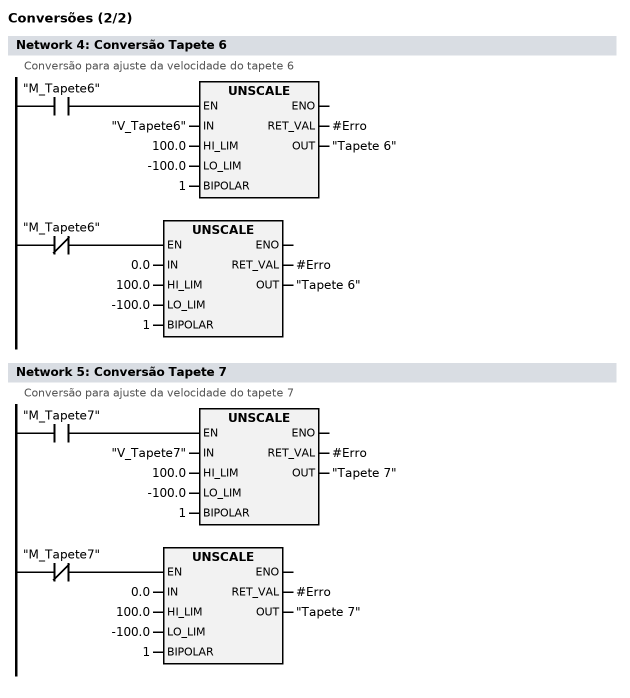
   IF "M_Tapete6" THEN
       #Erro := UNSCALE(IN := "V_Tapete6", HI_LIM := 100.0, LO_LIM := -100.0, BIPOLAR := 1, OUT => "Tapete 6");
   END_IF;
   IF NOT "M_Tapete6" THEN
       #Erro := UNSCALE(IN := 0.0, HI_LIM := 100.0, LO_LIM := -100.0, BIPOLAR := 1, OUT => "Tapete 6");
   END_IF;
END_REGION

REGION Network 5: Conversão Tapete 7
   // Conversão para ajuste da velocidade do tapete 7
   IF "M_Tapete7" THEN
       #Erro := UNSCALE(IN := "V_Tapete7", HI_LIM := 100.0, LO_LIM := -100.0, BIPOLAR := 1, OUT => "Tapete 7");
   END_IF;
   IF NOT "M_Tapete7" THEN
       #Erro := UNSCALE(IN := 0.0, HI_LIM := 100.0, LO_LIM := -100.0, BIPOLAR := 1, OUT => "Tapete 7");
   END_IF;
END_REGION
END_FUNCTION

FUNCTION "Controlo Secundário" : Void   // FC4, LAD
TITLE = Controlo Secundário
{ S7_Optimized_Access := 'TRUE' }
VERSION : 0.1
   VAR_TEMP
      "pulse 1" : Bool;
      "pulse 2" : Bool;
      "pulse 3" : Bool;
      "pulse 4" : Bool;
      "pulse 5" : Bool;
      "pulse 6" : Bool;
      "pulse 7" : Bool;
      "pulse 8" : Bool;
      "pulse 9" : Bool;
      "pulse 10" : Bool;
      "pulse 11" : Bool;
      "pulse 12" : Bool;
      "pulse 13" : Bool;
      "pulse 14" : Bool;
      "pulse 15" : Bool;
      "pulse 16" : Bool;
   END_VAR
   VAR_TEMP   // added for the SCL form of the ladder/FBD networks
      _w1 : Bool;
      _w2 : Bool;
   END_VAR
BEGIN

REGION Network 1: Move do posto inicial
   // Move 1 para atualizar o número do posto de armazenamento
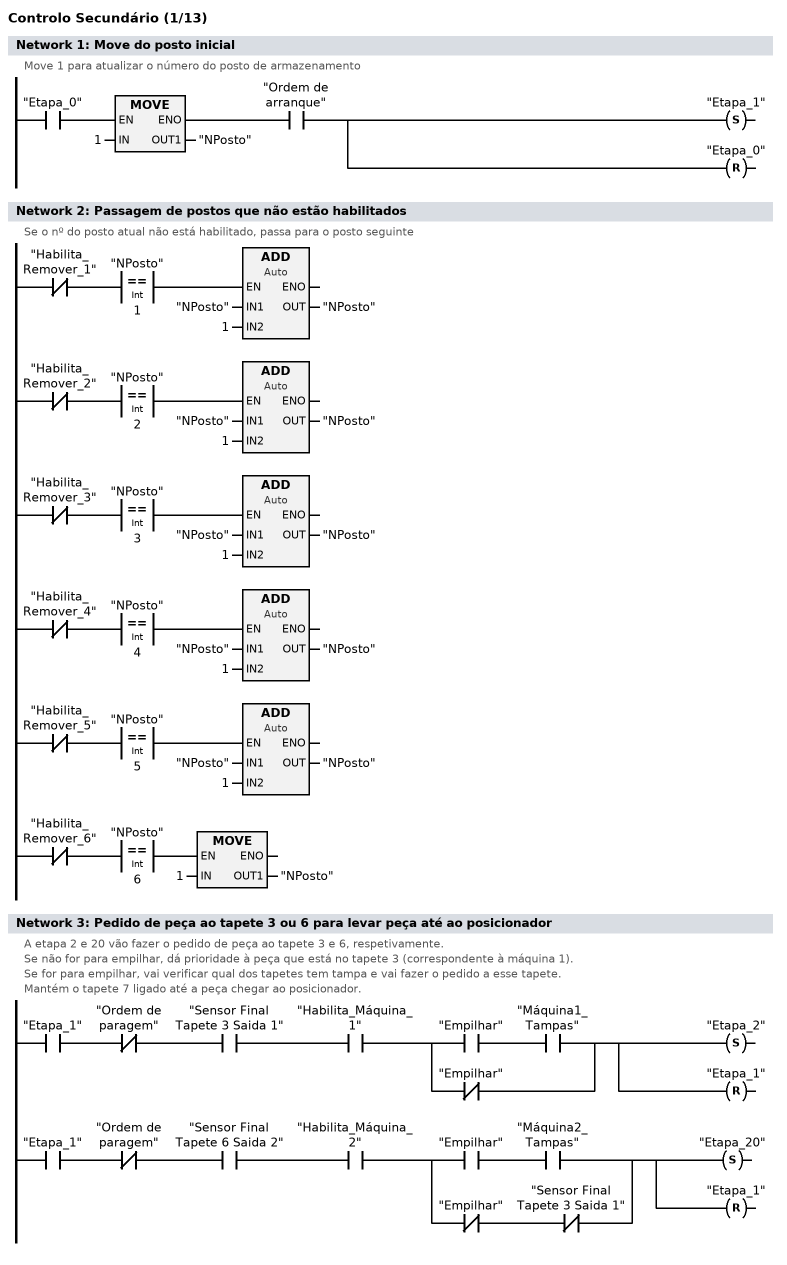
   RUNG wire#powerrail
      Contact( "Etapa_0" )
      Move(in := 1, out1 => "NPosto")
      Contact( "Ordem de arranque" )
      wire#w1
      S_Coil( "Etapa_1" )
   END_RUNG
   RUNG wire#w1
      R_Coil( "Etapa_0" )
   END_RUNG
   // the same network as SCL:
   IF "Etapa_0" THEN "NPosto" := 1; END_IF;
   IF "Etapa_0" AND "Ordem de arranque" THEN
       "Etapa_1" := TRUE;
       "Etapa_0" := FALSE;
   END_IF;
END_REGION

REGION Network 2: Passagem de postos que não estão habilitados
   // Se o nº do posto atual não está habilitado, passa para o posto seguinte
   RUNG wire#powerrail
      I_Contact( "Habilita_Remover_1" )
      { S7_Templates := "SrcType := Int" } EQ_Contact(in1 := "NPosto", in2 := 1)
      Add(in1 := "NPosto", in2 := 1, out => "NPosto")
   END_RUNG
   RUNG wire#powerrail
      I_Contact( "Habilita_Remover_2" )
      { S7_Templates := "SrcType := Int" } EQ_Contact(in1 := "NPosto", in2 := 2)
      Add(in1 := "NPosto", in2 := 1, out => "NPosto")
   END_RUNG
   RUNG wire#powerrail
      I_Contact( "Habilita_Remover_3" )
      { S7_Templates := "SrcType := Int" } EQ_Contact(in1 := "NPosto", in2 := 3)
      Add(in1 := "NPosto", in2 := 1, out => "NPosto")
   END_RUNG
   RUNG wire#powerrail
      I_Contact( "Habilita_Remover_4" )
      { S7_Templates := "SrcType := Int" } EQ_Contact(in1 := "NPosto", in2 := 4)
      Add(in1 := "NPosto", in2 := 1, out => "NPosto")
   END_RUNG
   RUNG wire#powerrail
      I_Contact( "Habilita_Remover_5" )
      { S7_Templates := "SrcType := Int" } EQ_Contact(in1 := "NPosto", in2 := 5)
      Add(in1 := "NPosto", in2 := 1, out => "NPosto")
   END_RUNG
   RUNG wire#powerrail
      I_Contact( "Habilita_Remover_6" )
      { S7_Templates := "SrcType := Int" } EQ_Contact(in1 := "NPosto", in2 := 6)
      Move(in := 1, out1 => "NPosto")
   END_RUNG
   // the same network as SCL:
   IF NOT "Habilita_Remover_1" AND ("NPosto" = 1) THEN "NPosto" := "NPosto" + 1; END_IF;
   IF NOT "Habilita_Remover_2" AND ("NPosto" = 2) THEN "NPosto" := "NPosto" + 1; END_IF;
   IF NOT "Habilita_Remover_3" AND ("NPosto" = 3) THEN "NPosto" := "NPosto" + 1; END_IF;
   IF NOT "Habilita_Remover_4" AND ("NPosto" = 4) THEN "NPosto" := "NPosto" + 1; END_IF;
   IF NOT "Habilita_Remover_5" AND ("NPosto" = 5) THEN "NPosto" := "NPosto" + 1; END_IF;
   IF NOT "Habilita_Remover_6" AND ("NPosto" = 6) THEN "NPosto" := 1; END_IF;
END_REGION

REGION Network 3: Pedido de peça ao tapete 3 ou 6 para levar peça até ao posicionador
   // A etapa 2 e 20 vão fazer o pedido de peça ao tapete 3 e 6, respetivamente.
   // Se não for para empilhar, dá prioridade à peça que está no tapete 3 (correspondente à máquina 1).
   // Se for para empilhar, vai verificar qual dos tapetes tem tampa e vai fazer o pedido a esse tapete.
   // Mantém o tapete 7 ligado até a peça chegar ao posicionador.
   RUNG wire#powerrail
      Contact( "Etapa_1" )
      I_Contact( "Ordem de paragem" )
      Contact( "Sensor Final Tapete 3 Saida 1" )
      Contact( "Habilita_Máquina_1" )
      wire#w1
      Contact( "Empilhar" )
      Contact( "Máquina1_Tampas" )
      wire#w2
      S_Coil( "Etapa_2" )
   END_RUNG
   RUNG wire#w1
      I_Contact( "Empilhar" )
   END_RUNG wire#w2
   RUNG wire#w2
      R_Coil( "Etapa_1" )
   END_RUNG
   RUNG wire#powerrail
      Contact( "Etapa_1" )
      I_Contact( "Ordem de paragem" )
      Contact( "Sensor Final Tapete 6 Saida 2" )
      Contact( "Habilita_Máquina_2" )
      wire#w3
      Contact( "Empilhar" )
      Contact( "Máquina2_Tampas" )
      wire#w4
      S_Coil( "Etapa_20" )
   END_RUNG
   RUNG wire#w3
      I_Contact( "Empilhar" )
      I_Contact( "Sensor Final Tapete 3 Saida 1" )
   END_RUNG wire#w4
   RUNG wire#w4
      R_Coil( "Etapa_1" )
   END_RUNG
   // the same network as SCL:
   IF "Etapa_1" AND NOT "Ordem de paragem" AND "Sensor Final Tapete 3 Saida 1" AND "Habilita_Máquina_1" AND (("Empilhar" AND "Máquina1_Tampas") OR NOT "Empilhar") THEN
       "Etapa_2" := TRUE;
       "Etapa_1" := FALSE;
   END_IF;
   IF "Etapa_1" AND NOT "Ordem de paragem" AND "Sensor Final Tapete 6 Saida 2" AND "Habilita_Máquina_2" AND (("Empilhar" AND "Máquina2_Tampas") OR (NOT "Empilhar" AND NOT "Sensor Final Tapete 3 Saida 1")) THEN
       "Etapa_20" := TRUE;
       "Etapa_1" := FALSE;
   END_IF;
END_REGION

REGION Network 4: Peça no posicionador
   // Quando a peça chega ao posicionador (sensor final tapete 7), vai fechar o grampo para centrar a peça
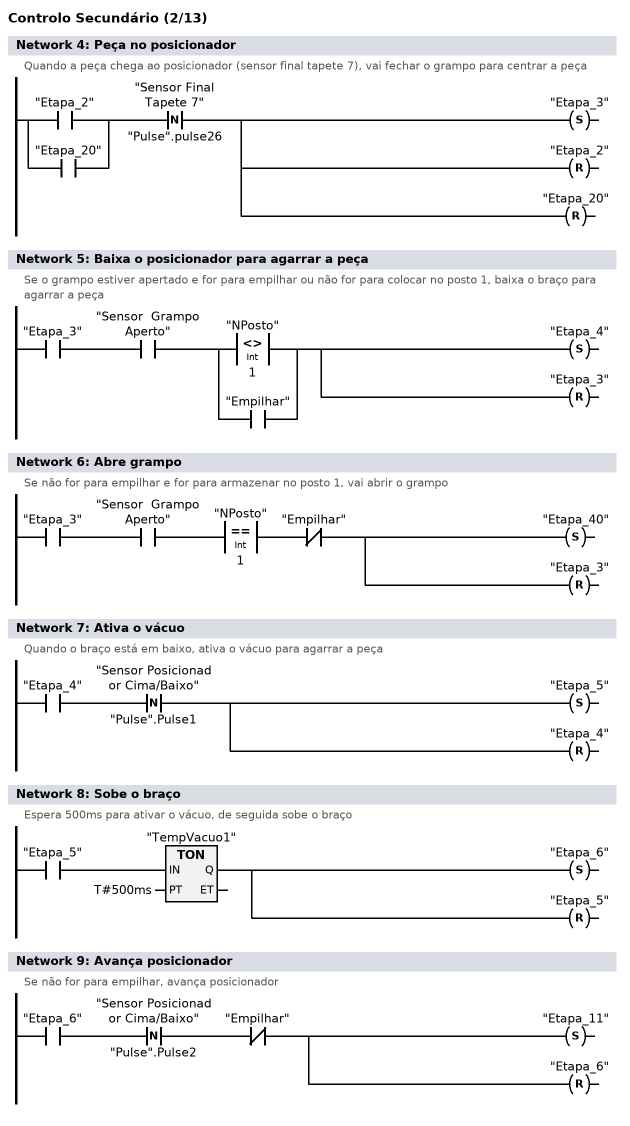
   RUNG wire#powerrail
      Contact( "Etapa_2" )
      wire#w1
      N_Contact(operand := "Sensor Final Tapete 7", bit := "Pulse".pulse26)
      wire#w2
      S_Coil( "Etapa_3" )
   END_RUNG
   RUNG wire#powerrail
      Contact( "Etapa_20" )
   END_RUNG wire#w1
   RUNG wire#w2
      R_Coil( "Etapa_2" )
   END_RUNG
   RUNG wire#w2
      R_Coil( "Etapa_20" )
   END_RUNG
   // the same network as SCL:
   #_w1 := ("Etapa_2" OR "Etapa_20") AND NOT "Sensor Final Tapete 7" AND "Pulse".pulse26;   // falling edge of "Sensor Final Tapete 7"
   "Pulse".pulse26 := "Sensor Final Tapete 7";
   IF #_w1 THEN
       "Etapa_3" := TRUE;
       "Etapa_2" := FALSE;
       "Etapa_20" := FALSE;
   END_IF;
END_REGION

REGION Network 5: Baixa o posicionador para agarrar a peça
   // Se o grampo estiver apertado e for para empilhar ou não for para colocar no posto 1, baixa o braço para agarrar a peça
   RUNG wire#powerrail
      Contact( "Etapa_3" )
      Contact( "Sensor  Grampo Aperto" )
      wire#w1
      { S7_Templates := "SrcType := Int" } NE_Contact(in1 := "NPosto", in2 := 1)
      wire#w2
      S_Coil( "Etapa_4" )
   END_RUNG
   RUNG wire#w1
      Contact( "Empilhar" )
   END_RUNG wire#w2
   RUNG wire#w2
      R_Coil( "Etapa_3" )
   END_RUNG
   // the same network as SCL:
   IF "Etapa_3" AND "Sensor  Grampo Aperto" AND (("NPosto" <> 1) OR "Empilhar") THEN
       "Etapa_4" := TRUE;
       "Etapa_3" := FALSE;
   END_IF;
END_REGION

REGION Network 6: Abre grampo
   // Se não for para empilhar e for para armazenar no posto 1, vai abrir o grampo
   RUNG wire#powerrail
      Contact( "Etapa_3" )
      Contact( "Sensor  Grampo Aperto" )
      { S7_Templates := "SrcType := Int" } EQ_Contact(in1 := "NPosto", in2 := 1)
      I_Contact( "Empilhar" )
      wire#w1
      S_Coil( "Etapa_40" )
   END_RUNG
   RUNG wire#w1
      R_Coil( "Etapa_3" )
   END_RUNG
   // the same network as SCL:
   IF "Etapa_3" AND "Sensor  Grampo Aperto" AND ("NPosto" = 1) AND NOT "Empilhar" THEN
       "Etapa_40" := TRUE;
       "Etapa_3" := FALSE;
   END_IF;
END_REGION

REGION Network 7: Ativa o vácuo
   // Quando o braço está em baixo, ativa o vácuo para agarrar a peça
   RUNG wire#powerrail
      Contact( "Etapa_4" )
      N_Contact(operand := "Sensor Posicionador Cima/Baixo", bit := "Pulse".Pulse1)
      wire#w1
      S_Coil( "Etapa_5" )
   END_RUNG
   RUNG wire#w1
      R_Coil( "Etapa_4" )
   END_RUNG
   // the same network as SCL:
   #_w1 := "Etapa_4" AND NOT "Sensor Posicionador Cima/Baixo" AND "Pulse".Pulse1;   // falling edge of "Sensor Posicionador Cima/Baixo"
   "Pulse".Pulse1 := "Sensor Posicionador Cima/Baixo";
   IF #_w1 THEN
       "Etapa_5" := TRUE;
       "Etapa_4" := FALSE;
   END_IF;
END_REGION

REGION Network 8: Sobe o braço
   // Espera 500ms para ativar o vácuo, de seguida sobe o braço
   "TempVacuo1".TON(IN := "Etapa_5", PT := T#500ms);
   IF "TempVacuo1".Q THEN
       "Etapa_6" := TRUE;
       "Etapa_5" := FALSE;
   END_IF;
END_REGION

REGION Network 9: Avança posicionador
   // Se não for para empilhar, avança posicionador
   RUNG wire#powerrail
      Contact( "Etapa_6" )
      N_Contact(operand := "Sensor Posicionador Cima/Baixo", bit := "Pulse".Pulse2)
      I_Contact( "Empilhar" )
      wire#w1
      S_Coil( "Etapa_11" )
   END_RUNG
   RUNG wire#w1
      R_Coil( "Etapa_6" )
   END_RUNG
   // the same network as SCL:
   #_w1 := "Etapa_6" AND NOT "Sensor Posicionador Cima/Baixo" AND "Pulse".Pulse2;   // falling edge of "Sensor Posicionador Cima/Baixo"
   "Pulse".Pulse2 := "Sensor Posicionador Cima/Baixo";
   IF #_w1 AND NOT "Empilhar" THEN
       "Etapa_11" := TRUE;
       "Etapa_6" := FALSE;
   END_IF;
END_REGION

REGION Network 10: Pedido da base
   // Quando é para empilhar e o braço chega acima, pede base ao tapete que tem a base, mantém o vácuo e liga o tapete 7
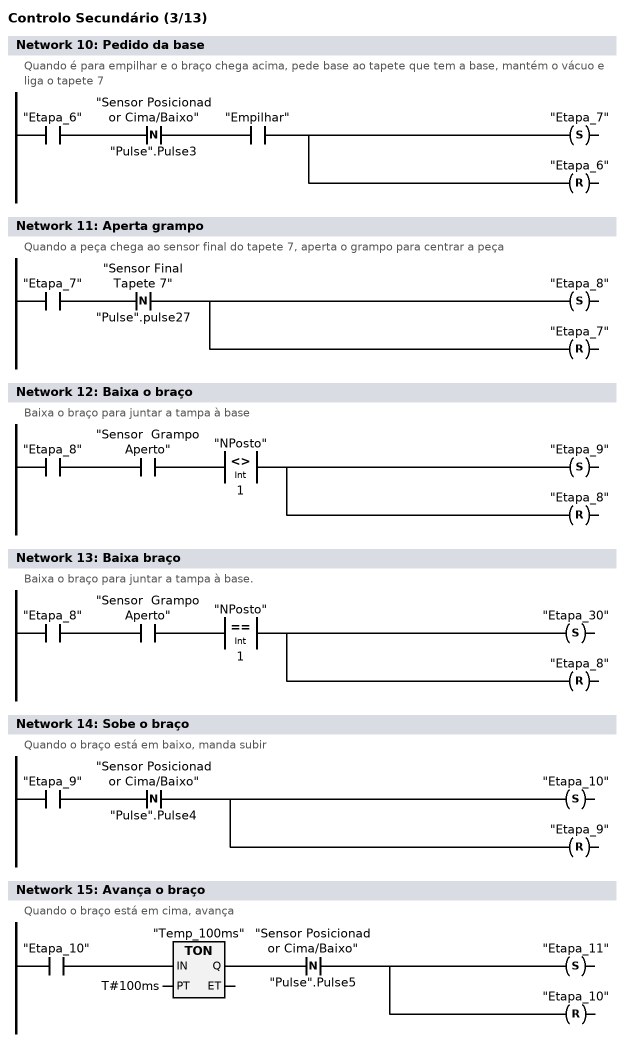
   RUNG wire#powerrail
      Contact( "Etapa_6" )
      N_Contact(operand := "Sensor Posicionador Cima/Baixo", bit := "Pulse".Pulse3)
      Contact( "Empilhar" )
      wire#w1
      S_Coil( "Etapa_7" )
   END_RUNG
   RUNG wire#w1
      R_Coil( "Etapa_6" )
   END_RUNG
   // the same network as SCL:
   #_w1 := "Etapa_6" AND NOT "Sensor Posicionador Cima/Baixo" AND "Pulse".Pulse3;   // falling edge of "Sensor Posicionador Cima/Baixo"
   "Pulse".Pulse3 := "Sensor Posicionador Cima/Baixo";
   IF #_w1 AND "Empilhar" THEN
       "Etapa_7" := TRUE;
       "Etapa_6" := FALSE;
   END_IF;
END_REGION

REGION Network 11: Aperta grampo
   // Quando a peça chega ao sensor final do tapete 7, aperta o grampo para centrar a peça
   RUNG wire#powerrail
      Contact( "Etapa_7" )
      N_Contact(operand := "Sensor Final Tapete 7", bit := "Pulse".pulse27)
      wire#w1
      S_Coil( "Etapa_8" )
   END_RUNG
   RUNG wire#w1
      R_Coil( "Etapa_7" )
   END_RUNG
   // the same network as SCL:
   #_w1 := "Etapa_7" AND NOT "Sensor Final Tapete 7" AND "Pulse".pulse27;   // falling edge of "Sensor Final Tapete 7"
   "Pulse".pulse27 := "Sensor Final Tapete 7";
   IF #_w1 THEN
       "Etapa_8" := TRUE;
       "Etapa_7" := FALSE;
   END_IF;
END_REGION

REGION Network 12: Baixa o braço
   // Baixa o braço para juntar a tampa à base
   RUNG wire#powerrail
      Contact( "Etapa_8" )
      Contact( "Sensor  Grampo Aperto" )
      { S7_Templates := "SrcType := Int" } NE_Contact(in1 := "NPosto", in2 := 1)
      wire#w1
      S_Coil( "Etapa_9" )
   END_RUNG
   RUNG wire#w1
      R_Coil( "Etapa_8" )
   END_RUNG
   // the same network as SCL:
   IF "Etapa_8" AND "Sensor  Grampo Aperto" AND ("NPosto" <> 1) THEN
       "Etapa_9" := TRUE;
       "Etapa_8" := FALSE;
   END_IF;
END_REGION

REGION Network 13: Baixa braço
   // Baixa o braço para juntar a tampa à base.
   RUNG wire#powerrail
      Contact( "Etapa_8" )
      Contact( "Sensor  Grampo Aperto" )
      { S7_Templates := "SrcType := Int" } EQ_Contact(in1 := "NPosto", in2 := 1)
      wire#w1
      S_Coil( "Etapa_30" )
   END_RUNG
   RUNG wire#w1
      R_Coil( "Etapa_8" )
   END_RUNG
   // the same network as SCL:
   IF "Etapa_8" AND "Sensor  Grampo Aperto" AND ("NPosto" = 1) THEN
       "Etapa_30" := TRUE;
       "Etapa_8" := FALSE;
   END_IF;
END_REGION

REGION Network 14: Sobe o braço
   // Quando o braço está em baixo, manda subir
   RUNG wire#powerrail
      Contact( "Etapa_9" )
      N_Contact(operand := "Sensor Posicionador Cima/Baixo", bit := "Pulse".Pulse4)
      wire#w1
      S_Coil( "Etapa_10" )
   END_RUNG
   RUNG wire#w1
      R_Coil( "Etapa_9" )
   END_RUNG
   // the same network as SCL:
   #_w1 := "Etapa_9" AND NOT "Sensor Posicionador Cima/Baixo" AND "Pulse".Pulse4;   // falling edge of "Sensor Posicionador Cima/Baixo"
   "Pulse".Pulse4 := "Sensor Posicionador Cima/Baixo";
   IF #_w1 THEN
       "Etapa_10" := TRUE;
       "Etapa_9" := FALSE;
   END_IF;
END_REGION

REGION Network 15: Avança o braço
   // Quando o braço está em cima, avança
   "Temp_100ms".TON(IN := "Etapa_10", PT := T#100ms);
   #_w1 := "Temp_100ms".Q AND NOT "Sensor Posicionador Cima/Baixo" AND "Pulse".Pulse5;   // falling edge of "Sensor Posicionador Cima/Baixo"
   "Pulse".Pulse5 := "Sensor Posicionador Cima/Baixo";
   IF #_w1 THEN
       "Etapa_11" := TRUE;
       "Etapa_10" := FALSE;
   END_IF;
END_REGION

REGION Network 16: Baixa o braço
   // Quando o braço chega à frente, baixa o braço
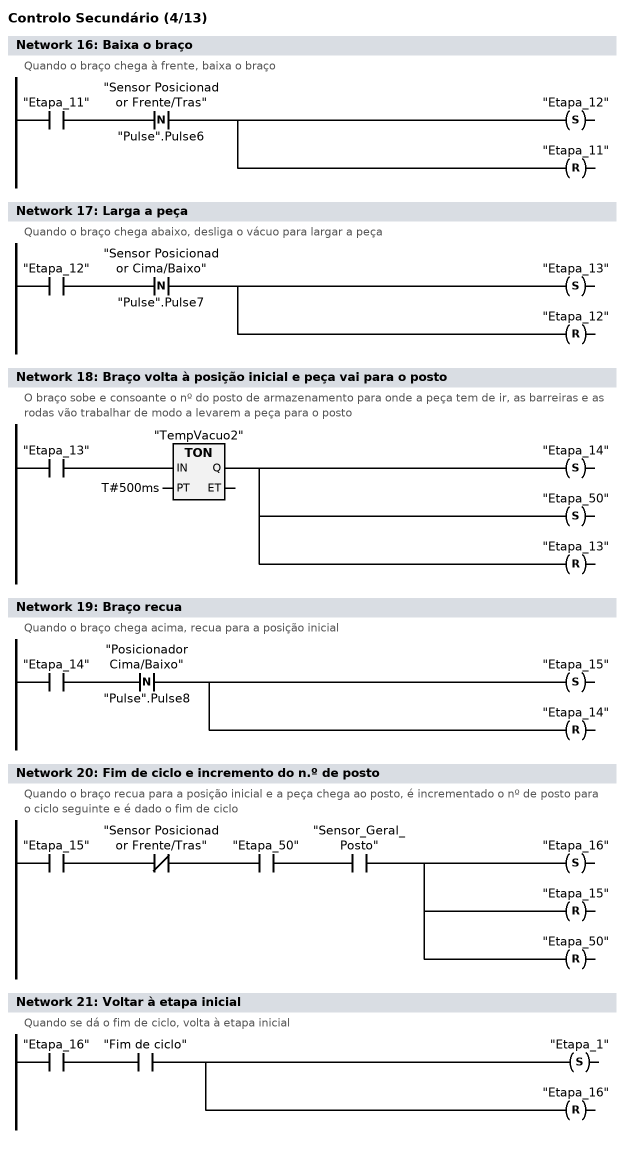
   RUNG wire#powerrail
      Contact( "Etapa_11" )
      N_Contact(operand := "Sensor Posicionador Frente/Tras", bit := "Pulse".Pulse6)
      wire#w1
      S_Coil( "Etapa_12" )
   END_RUNG
   RUNG wire#w1
      R_Coil( "Etapa_11" )
   END_RUNG
   // the same network as SCL:
   #_w1 := "Etapa_11" AND NOT "Sensor Posicionador Frente/Tras" AND "Pulse".Pulse6;   // falling edge of "Sensor Posicionador Frente/Tras"
   "Pulse".Pulse6 := "Sensor Posicionador Frente/Tras";
   IF #_w1 THEN
       "Etapa_12" := TRUE;
       "Etapa_11" := FALSE;
   END_IF;
END_REGION

REGION Network 17: Larga a peça
   // Quando o braço chega abaixo, desliga o vácuo para largar a peça
   RUNG wire#powerrail
      Contact( "Etapa_12" )
      N_Contact(operand := "Sensor Posicionador Cima/Baixo", bit := "Pulse".Pulse7)
      wire#w1
      S_Coil( "Etapa_13" )
   END_RUNG
   RUNG wire#w1
      R_Coil( "Etapa_12" )
   END_RUNG
   // the same network as SCL:
   #_w1 := "Etapa_12" AND NOT "Sensor Posicionador Cima/Baixo" AND "Pulse".Pulse7;   // falling edge of "Sensor Posicionador Cima/Baixo"
   "Pulse".Pulse7 := "Sensor Posicionador Cima/Baixo";
   IF #_w1 THEN
       "Etapa_13" := TRUE;
       "Etapa_12" := FALSE;
   END_IF;
END_REGION

REGION Network 18: Braço volta à posição inicial e peça vai para o posto
   // O braço sobe e consoante o nº do posto de armazenamento para onde a peça tem de ir, as barreiras e as rodas vão trabalhar de modo a levarem a peça para o posto
   "TempVacuo2".TON(IN := "Etapa_13", PT := T#500ms);
   IF "TempVacuo2".Q THEN
       "Etapa_14" := TRUE;
       "Etapa_50" := TRUE;
       "Etapa_13" := FALSE;
   END_IF;
END_REGION

REGION Network 19: Braço recua
   // Quando o braço chega acima, recua para a posição inicial
   RUNG wire#powerrail
      Contact( "Etapa_14" )
      N_Contact(operand := "Posicionador Cima/Baixo", bit := "Pulse".Pulse8)
      wire#w1
      S_Coil( "Etapa_15" )
   END_RUNG
   RUNG wire#w1
      R_Coil( "Etapa_14" )
   END_RUNG
   // the same network as SCL:
   #_w1 := "Etapa_14" AND NOT "Posicionador Cima/Baixo" AND "Pulse".Pulse8;   // falling edge of "Posicionador Cima/Baixo"
   "Pulse".Pulse8 := "Posicionador Cima/Baixo";
   IF #_w1 THEN
       "Etapa_15" := TRUE;
       "Etapa_14" := FALSE;
   END_IF;
END_REGION

REGION Network 20: Fim de ciclo e incremento do n.º de posto
   // Quando o braço recua para a posição inicial e a peça chega ao posto, é incrementado o nº de posto para o ciclo seguinte e é dado o fim de ciclo
   RUNG wire#powerrail
      Contact( "Etapa_15" )
      I_Contact( "Sensor Posicionador Frente/Tras" )
      Contact( "Etapa_50" )
      Contact( "Sensor_Geral_Posto" )
      wire#w1
      S_Coil( "Etapa_16" )
   END_RUNG
   RUNG wire#w1
      R_Coil( "Etapa_15" )
   END_RUNG
   RUNG wire#w1
      R_Coil( "Etapa_50" )
   END_RUNG
   // the same network as SCL:
   IF "Etapa_15" AND NOT "Sensor Posicionador Frente/Tras" AND "Etapa_50" AND "Sensor_Geral_Posto" THEN
       "Etapa_16" := TRUE;
   END_IF;
   #_w1 := "Etapa_15" AND NOT "Sensor Posicionador Frente/Tras" AND "Etapa_50" AND "Sensor_Geral_Posto";
   IF #_w1 THEN
       "Etapa_15" := FALSE;
       "Etapa_50" := FALSE;
   END_IF;
END_REGION

REGION Network 21: Voltar à etapa inicial
   // Quando se dá o fim de ciclo, volta à etapa inicial
   RUNG wire#powerrail
      Contact( "Etapa_16" )
      Contact( "Fim de ciclo" )
      wire#w1
      S_Coil( "Etapa_1" )
   END_RUNG
   RUNG wire#w1
      R_Coil( "Etapa_16" )
   END_RUNG
   // the same network as SCL:
   IF "Etapa_16" AND "Fim de ciclo" THEN
       "Etapa_1" := TRUE;
       "Etapa_16" := FALSE;
   END_IF;
END_REGION

REGION Network 22: Desliga o vácuo e sobe o braço
   // Quando o braço chega abaixo, desliga o vácuo para largar a peça e sobe o braço para a posição inicial
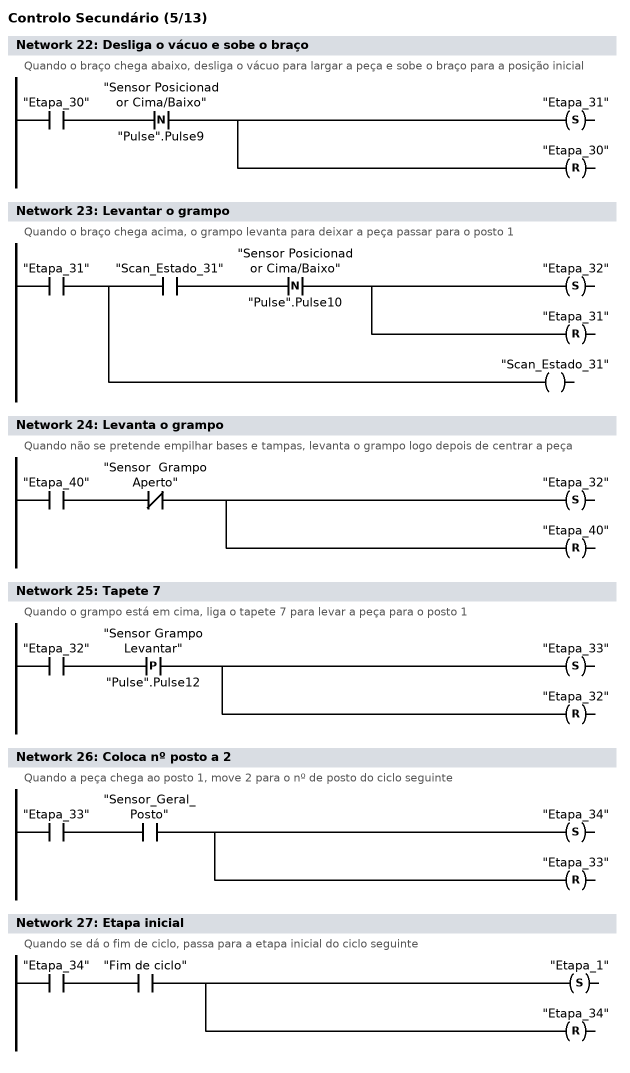
   RUNG wire#powerrail
      Contact( "Etapa_30" )
      N_Contact(operand := "Sensor Posicionador Cima/Baixo", bit := "Pulse".Pulse9)
      wire#w1
      S_Coil( "Etapa_31" )
   END_RUNG
   RUNG wire#w1
      R_Coil( "Etapa_30" )
   END_RUNG
   // the same network as SCL:
   #_w1 := "Etapa_30" AND NOT "Sensor Posicionador Cima/Baixo" AND "Pulse".Pulse9;   // falling edge of "Sensor Posicionador Cima/Baixo"
   "Pulse".Pulse9 := "Sensor Posicionador Cima/Baixo";
   IF #_w1 THEN
       "Etapa_31" := TRUE;
       "Etapa_30" := FALSE;
   END_IF;
END_REGION

REGION Network 23: Levantar o grampo
   // Quando o braço chega acima, o grampo levanta para deixar a peça passar para o posto 1
   RUNG wire#powerrail
      Contact( "Etapa_31" )
      wire#w1
      Contact( "Scan_Estado_31" )
      N_Contact(operand := "Sensor Posicionador Cima/Baixo", bit := "Pulse".Pulse10)
      wire#w2
      S_Coil( "Etapa_32" )
   END_RUNG
   RUNG wire#w2
      R_Coil( "Etapa_31" )
   END_RUNG
   RUNG wire#w1
      Coil( "Scan_Estado_31" )
   END_RUNG
   // the same network as SCL:
   #_w1 := "Etapa_31" AND "Scan_Estado_31" AND NOT "Sensor Posicionador Cima/Baixo" AND "Pulse".Pulse10;   // falling edge of "Sensor Posicionador Cima/Baixo"
   "Pulse".Pulse10 := "Sensor Posicionador Cima/Baixo";
   IF #_w1 THEN "Etapa_32" := TRUE; END_IF;
   #_w2 := "Etapa_31";
   IF #_w1 THEN "Etapa_31" := FALSE; END_IF;
   "Scan_Estado_31" := #_w2;
END_REGION

REGION Network 24: Levanta o grampo
   // Quando não se pretende empilhar bases e tampas, levanta o grampo logo depois de centrar a peça
   RUNG wire#powerrail
      Contact( "Etapa_40" )
      I_Contact( "Sensor  Grampo Aperto" )
      wire#w1
      S_Coil( "Etapa_32" )
   END_RUNG
   RUNG wire#w1
      R_Coil( "Etapa_40" )
   END_RUNG
   // the same network as SCL:
   IF "Etapa_40" AND NOT "Sensor  Grampo Aperto" THEN
       "Etapa_32" := TRUE;
       "Etapa_40" := FALSE;
   END_IF;
END_REGION

REGION Network 25: Tapete 7
   // Quando o grampo está em cima, liga o tapete 7 para levar a peça para o posto 1
   RUNG wire#powerrail
      Contact( "Etapa_32" )
      P_Contact(operand := "Sensor Grampo Levantar", bit := "Pulse".Pulse12)
      wire#w1
      S_Coil( "Etapa_33" )
   END_RUNG
   RUNG wire#w1
      R_Coil( "Etapa_32" )
   END_RUNG
   // the same network as SCL:
   #_w1 := "Etapa_32" AND "Sensor Grampo Levantar" AND NOT "Pulse".Pulse12;   // rising edge of "Sensor Grampo Levantar"
   "Pulse".Pulse12 := "Sensor Grampo Levantar";
   IF #_w1 THEN
       "Etapa_33" := TRUE;
       "Etapa_32" := FALSE;
   END_IF;
END_REGION

REGION Network 26: Coloca nº posto a 2
   // Quando a peça chega ao posto 1, move 2 para o nº de posto do ciclo seguinte
   RUNG wire#powerrail
      Contact( "Etapa_33" )
      Contact( "Sensor_Geral_Posto" )
      wire#w1
      S_Coil( "Etapa_34" )
   END_RUNG
   RUNG wire#w1
      R_Coil( "Etapa_33" )
   END_RUNG
   // the same network as SCL:
   IF "Etapa_33" AND "Sensor_Geral_Posto" THEN
       "Etapa_34" := TRUE;
       "Etapa_33" := FALSE;
   END_IF;
END_REGION

REGION Network 27: Etapa inicial
   // Quando se dá o fim de ciclo, passa para a etapa inicial do ciclo seguinte
   RUNG wire#powerrail
      Contact( "Etapa_34" )
      Contact( "Fim de ciclo" )
      wire#w1
      S_Coil( "Etapa_1" )
   END_RUNG
   RUNG wire#w1
      R_Coil( "Etapa_34" )
   END_RUNG
   // the same network as SCL:
   IF "Etapa_34" AND "Fim de ciclo" THEN
       "Etapa_1" := TRUE;
       "Etapa_34" := FALSE;
   END_IF;
END_REGION

REGION Network 28: Bit geral dos sensores de saida posto
   // Quando a peça passa no sensor do posto de saida selecionado, ativa este bit
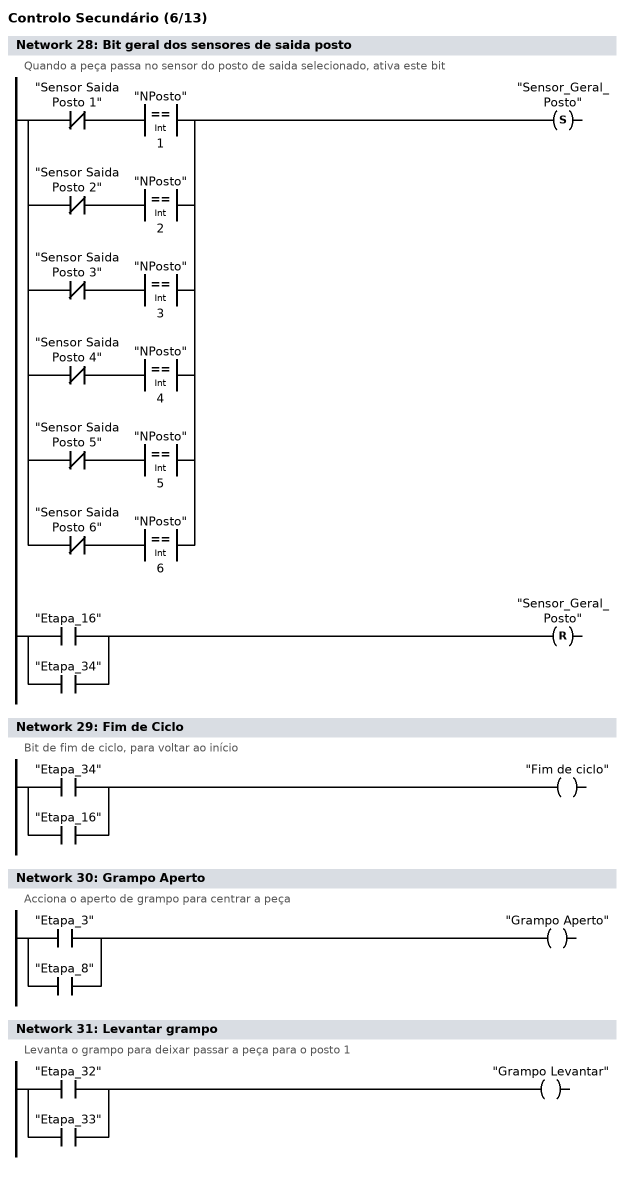
   RUNG wire#powerrail
      I_Contact( "Sensor Saida Posto 1" )
      { S7_Templates := "SrcType := Int" } EQ_Contact(in1 := "NPosto", in2 := 1)
      wire#w1
      S_Coil( "Sensor_Geral_Posto" )
   END_RUNG
   RUNG wire#powerrail
      I_Contact( "Sensor Saida Posto 2" )
      { S7_Templates := "SrcType := Int" } EQ_Contact(in1 := "NPosto", in2 := 2)
   END_RUNG wire#w1
   RUNG wire#powerrail
      I_Contact( "Sensor Saida Posto 3" )
      { S7_Templates := "SrcType := Int" } EQ_Contact(in1 := "NPosto", in2 := 3)
   END_RUNG wire#w1
   RUNG wire#powerrail
      I_Contact( "Sensor Saida Posto 4" )
      { S7_Templates := "SrcType := Int" } EQ_Contact(in1 := "NPosto", in2 := 4)
   END_RUNG wire#w1
   RUNG wire#powerrail
      I_Contact( "Sensor Saida Posto 5" )
      { S7_Templates := "SrcType := Int" } EQ_Contact(in1 := "NPosto", in2 := 5)
   END_RUNG wire#w1
   RUNG wire#powerrail
      I_Contact( "Sensor Saida Posto 6" )
      { S7_Templates := "SrcType := Int" } EQ_Contact(in1 := "NPosto", in2 := 6)
   END_RUNG wire#w1
   RUNG wire#powerrail
      Contact( "Etapa_16" )
      wire#w2
      R_Coil( "Sensor_Geral_Posto" )
   END_RUNG
   RUNG wire#powerrail
      Contact( "Etapa_34" )
   END_RUNG wire#w2
   // the same network as SCL:
   IF (NOT "Sensor Saida Posto 1" AND ("NPosto" = 1)) OR (NOT "Sensor Saida Posto 2" AND ("NPosto" = 2)) OR (NOT "Sensor Saida Posto 3" AND ("NPosto" = 3)) OR (NOT "Sensor Saida Posto 4" AND ("NPosto" = 4)) OR (NOT "Sensor Saida Posto 5" AND ("NPosto" = 5)) OR (NOT "Sensor Saida Posto 6" AND ("NPosto" = 6)) THEN
       "Sensor_Geral_Posto" := TRUE;
   END_IF;
   IF "Etapa_16" OR "Etapa_34" THEN "Sensor_Geral_Posto" := FALSE; END_IF;
END_REGION

REGION Network 29: Fim de Ciclo
   // Bit de fim de ciclo, para voltar ao início
   RUNG wire#powerrail
      Contact( "Etapa_34" )
      wire#w1
      Coil( "Fim de ciclo" )
   END_RUNG
   RUNG wire#powerrail
      Contact( "Etapa_16" )
   END_RUNG wire#w1
   // the same network as SCL:
   "Fim de ciclo" := "Etapa_34" OR "Etapa_16";
END_REGION

REGION Network 30: Grampo Aperto
   // Acciona o aperto de grampo para centrar a peça
   RUNG wire#powerrail
      Contact( "Etapa_3" )
      wire#w1
      Coil( "Grampo Aperto" )
   END_RUNG
   RUNG wire#powerrail
      Contact( "Etapa_8" )
   END_RUNG wire#w1
   // the same network as SCL:
   "Grampo Aperto" := "Etapa_3" OR "Etapa_8";
END_REGION

REGION Network 31: Levantar grampo
   // Levanta o grampo para deixar passar a peça para o posto 1
   RUNG wire#powerrail
      Contact( "Etapa_32" )
      wire#w1
      Coil( "Grampo Levantar" )
   END_RUNG
   RUNG wire#powerrail
      Contact( "Etapa_33" )
   END_RUNG wire#w1
   // the same network as SCL:
   "Grampo Levantar" := "Etapa_32" OR "Etapa_33";
END_REGION

REGION Network 32: Baixa Braço
   // Baixa o braço para agarrar e largar a peça
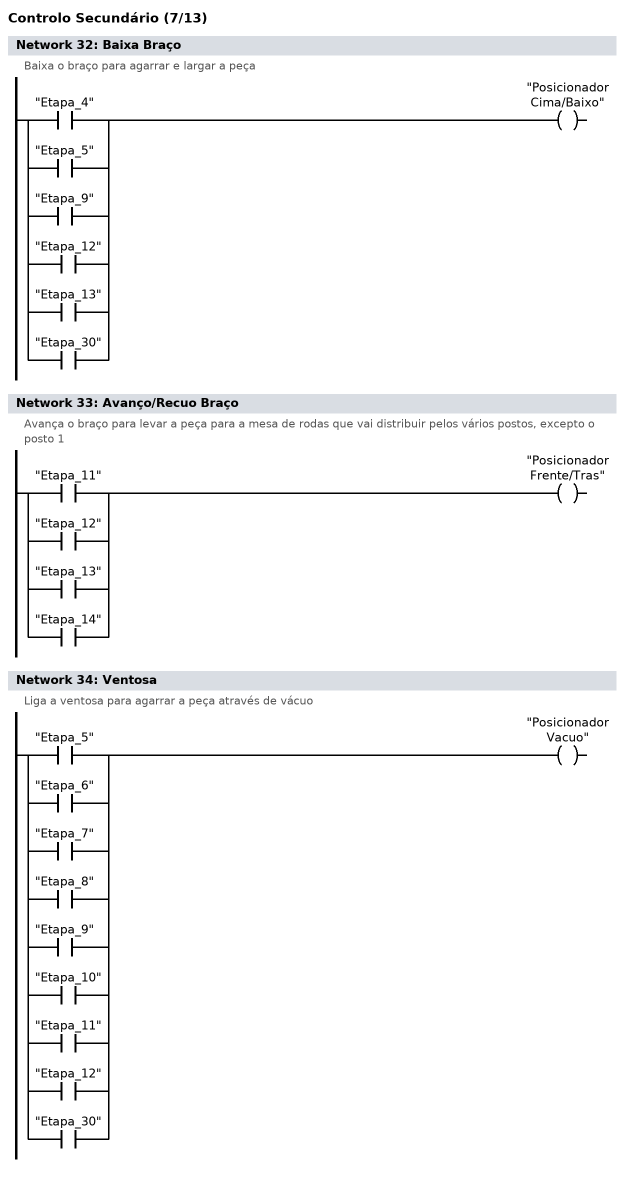
   RUNG wire#powerrail
      Contact( "Etapa_4" )
      wire#w1
      Coil( "Posicionador Cima/Baixo" )
   END_RUNG
   RUNG wire#powerrail
      Contact( "Etapa_5" )
   END_RUNG wire#w1
   RUNG wire#powerrail
      Contact( "Etapa_9" )
   END_RUNG wire#w1
   RUNG wire#powerrail
      Contact( "Etapa_12" )
   END_RUNG wire#w1
   RUNG wire#powerrail
      Contact( "Etapa_13" )
   END_RUNG wire#w1
   RUNG wire#powerrail
      Contact( "Etapa_30" )
   END_RUNG wire#w1
   // the same network as SCL:
   "Posicionador Cima/Baixo" := "Etapa_4" OR "Etapa_5" OR "Etapa_9" OR "Etapa_12" OR "Etapa_13" OR "Etapa_30";
END_REGION

REGION Network 33: Avanço/Recuo Braço
   // Avança o braço para levar a peça para a mesa de rodas que vai distribuir pelos vários postos, excepto o posto 1
   RUNG wire#powerrail
      Contact( "Etapa_11" )
      wire#w1
      Coil( "Posicionador Frente/Tras" )
   END_RUNG
   RUNG wire#powerrail
      Contact( "Etapa_12" )
   END_RUNG wire#w1
   RUNG wire#powerrail
      Contact( "Etapa_13" )
   END_RUNG wire#w1
   RUNG wire#powerrail
      Contact( "Etapa_14" )
   END_RUNG wire#w1
   // the same network as SCL:
   "Posicionador Frente/Tras" := "Etapa_11" OR "Etapa_12" OR "Etapa_13" OR "Etapa_14";
END_REGION

REGION Network 34: Ventosa
   // Liga a ventosa para agarrar a peça através de vácuo
   RUNG wire#powerrail
      Contact( "Etapa_5" )
      wire#w1
      Coil( "Posicionador Vacuo" )
   END_RUNG
   RUNG wire#powerrail
      Contact( "Etapa_6" )
   END_RUNG wire#w1
   RUNG wire#powerrail
      Contact( "Etapa_7" )
   END_RUNG wire#w1
   RUNG wire#powerrail
      Contact( "Etapa_8" )
   END_RUNG wire#w1
   RUNG wire#powerrail
      Contact( "Etapa_9" )
   END_RUNG wire#w1
   RUNG wire#powerrail
      Contact( "Etapa_10" )
   END_RUNG wire#w1
   RUNG wire#powerrail
      Contact( "Etapa_11" )
   END_RUNG wire#w1
   RUNG wire#powerrail
      Contact( "Etapa_12" )
   END_RUNG wire#w1
   RUNG wire#powerrail
      Contact( "Etapa_30" )
   END_RUNG wire#w1
   // the same network as SCL:
   "Posicionador Vacuo" := "Etapa_5" OR "Etapa_6" OR "Etapa_7" OR "Etapa_8" OR "Etapa_9" OR "Etapa_10" OR "Etapa_11" OR "Etapa_12" OR "Etapa_30";
END_REGION

REGION Network 35: Tapete 7
   // Liga o tapete 7
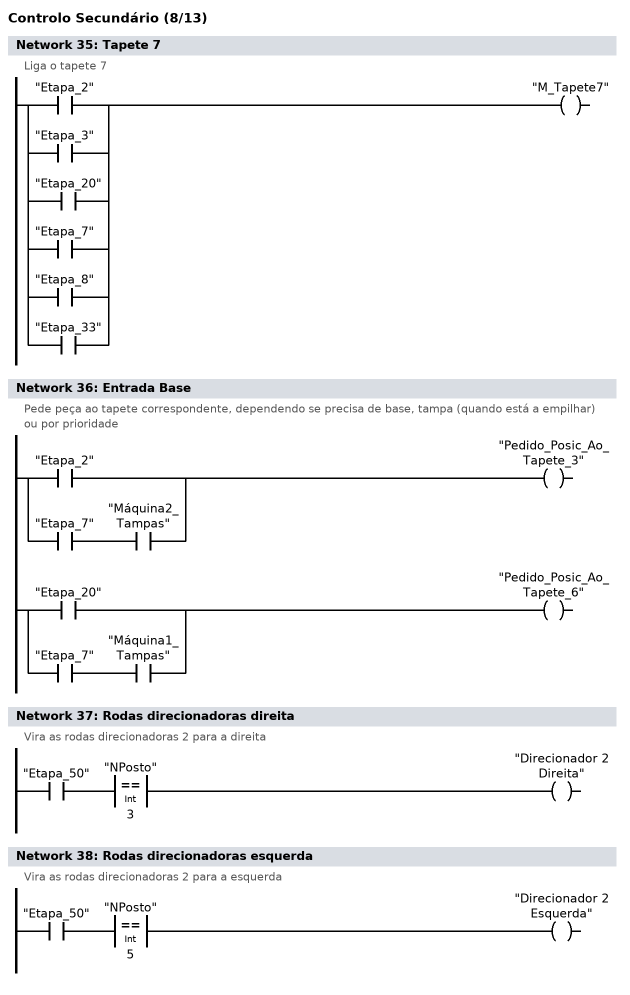
   RUNG wire#powerrail
      Contact( "Etapa_2" )
      wire#w1
      Coil( "M_Tapete7" )
   END_RUNG
   RUNG wire#powerrail
      Contact( "Etapa_3" )
   END_RUNG wire#w1
   RUNG wire#powerrail
      Contact( "Etapa_20" )
   END_RUNG wire#w1
   RUNG wire#powerrail
      Contact( "Etapa_7" )
   END_RUNG wire#w1
   RUNG wire#powerrail
      Contact( "Etapa_8" )
   END_RUNG wire#w1
   RUNG wire#powerrail
      Contact( "Etapa_33" )
   END_RUNG wire#w1
   // the same network as SCL:
   "M_Tapete7" := "Etapa_2" OR "Etapa_3" OR "Etapa_20" OR "Etapa_7" OR "Etapa_8" OR "Etapa_33";
END_REGION

REGION Network 36: Entrada Base
   // Pede peça ao tapete correspondente, dependendo se precisa de base, tampa (quando está a empilhar) ou por prioridade
   RUNG wire#powerrail
      Contact( "Etapa_2" )
      wire#w1
      Coil( "Pedido_Posic_Ao_Tapete_3" )
   END_RUNG
   RUNG wire#powerrail
      Contact( "Etapa_7" )
      Contact( "Máquina2_Tampas" )
   END_RUNG wire#w1
   RUNG wire#powerrail
      Contact( "Etapa_20" )
      wire#w2
      Coil( "Pedido_Posic_Ao_Tapete_6" )
   END_RUNG
   RUNG wire#powerrail
      Contact( "Etapa_7" )
      Contact( "Máquina1_Tampas" )
   END_RUNG wire#w2
   // the same network as SCL:
   "Pedido_Posic_Ao_Tapete_3" := "Etapa_2" OR ("Etapa_7" AND "Máquina2_Tampas");
   "Pedido_Posic_Ao_Tapete_6" := "Etapa_20" OR ("Etapa_7" AND "Máquina1_Tampas");
END_REGION

REGION Network 37: Rodas direcionadoras direita
   // Vira as rodas direcionadoras 2 para a direita
   RUNG wire#powerrail
      Contact( "Etapa_50" )
      { S7_Templates := "SrcType := Int" } EQ_Contact(in1 := "NPosto", in2 := 3)
      Coil( "Direcionador 2 Direita" )
   END_RUNG
   // the same network as SCL:
   "Direcionador 2 Direita" := "Etapa_50" AND ("NPosto" = 3);
END_REGION

REGION Network 38: Rodas direcionadoras esquerda
   // Vira as rodas direcionadoras 2 para a esquerda
   RUNG wire#powerrail
      Contact( "Etapa_50" )
      { S7_Templates := "SrcType := Int" } EQ_Contact(in1 := "NPosto", in2 := 5)
      Coil( "Direcionador 2 Esquerda" )
   END_RUNG
   // the same network as SCL:
   "Direcionador 2 Esquerda" := "Etapa_50" AND ("NPosto" = 5);
END_REGION

REGION Network 39: Rodas direcionadoras
   // Liga as rodas direcionadoras
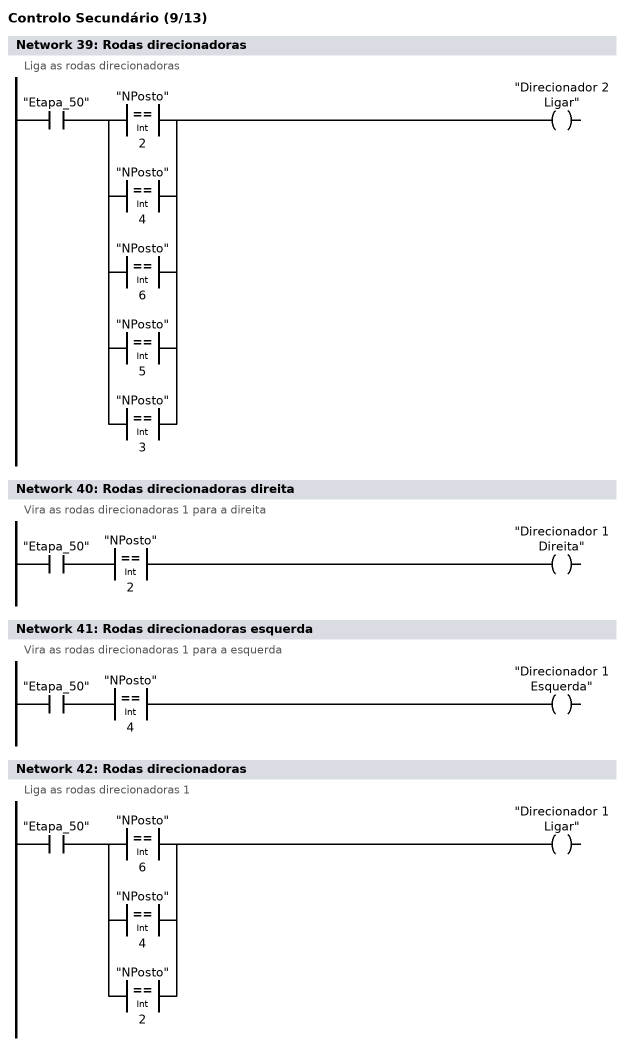
   RUNG wire#powerrail
      Contact( "Etapa_50" )
      wire#w1
      { S7_Templates := "SrcType := Int" } EQ_Contact(in1 := "NPosto", in2 := 2)
      wire#w2
      Coil( "Direcionador 2 Ligar" )
   END_RUNG
   RUNG wire#w1
      { S7_Templates := "SrcType := Int" } EQ_Contact(in1 := "NPosto", in2 := 4)
   END_RUNG wire#w2
   RUNG wire#w1
      { S7_Templates := "SrcType := Int" } EQ_Contact(in1 := "NPosto", in2 := 6)
   END_RUNG wire#w2
   RUNG wire#w1
      { S7_Templates := "SrcType := Int" } EQ_Contact(in1 := "NPosto", in2 := 5)
   END_RUNG wire#w2
   RUNG wire#w1
      { S7_Templates := "SrcType := Int" } EQ_Contact(in1 := "NPosto", in2 := 3)
   END_RUNG wire#w2
   // the same network as SCL:
   "Direcionador 2 Ligar" := "Etapa_50" AND (("NPosto" = 2) OR ("NPosto" = 4) OR ("NPosto" = 6) OR ("NPosto" = 5) OR ("NPosto" = 3));
END_REGION

REGION Network 40: Rodas direcionadoras direita
   // Vira as rodas direcionadoras 1 para a direita
   RUNG wire#powerrail
      Contact( "Etapa_50" )
      { S7_Templates := "SrcType := Int" } EQ_Contact(in1 := "NPosto", in2 := 2)
      Coil( "Direcionador 1 Direita" )
   END_RUNG
   // the same network as SCL:
   "Direcionador 1 Direita" := "Etapa_50" AND ("NPosto" = 2);
END_REGION

REGION Network 41: Rodas direcionadoras esquerda
   // Vira as rodas direcionadoras 1 para a esquerda
   RUNG wire#powerrail
      Contact( "Etapa_50" )
      { S7_Templates := "SrcType := Int" } EQ_Contact(in1 := "NPosto", in2 := 4)
      Coil( "Direcionador 1 Esquerda" )
   END_RUNG
   // the same network as SCL:
   "Direcionador 1 Esquerda" := "Etapa_50" AND ("NPosto" = 4);
END_REGION

REGION Network 42: Rodas direcionadoras
   // Liga as rodas direcionadoras 1
   RUNG wire#powerrail
      Contact( "Etapa_50" )
      wire#w1
      { S7_Templates := "SrcType := Int" } EQ_Contact(in1 := "NPosto", in2 := 6)
      wire#w2
      Coil( "Direcionador 1 Ligar" )
   END_RUNG
   RUNG wire#w1
      { S7_Templates := "SrcType := Int" } EQ_Contact(in1 := "NPosto", in2 := 4)
   END_RUNG wire#w2
   RUNG wire#w1
      { S7_Templates := "SrcType := Int" } EQ_Contact(in1 := "NPosto", in2 := 2)
   END_RUNG wire#w2
   // the same network as SCL:
   "Direcionador 1 Ligar" := "Etapa_50" AND (("NPosto" = 6) OR ("NPosto" = 4) OR ("NPosto" = 2));
END_REGION

REGION Network 43: Barreira posto 2 e 4
   // Sobe a barreira que leva a peça para os postos 2 e 4
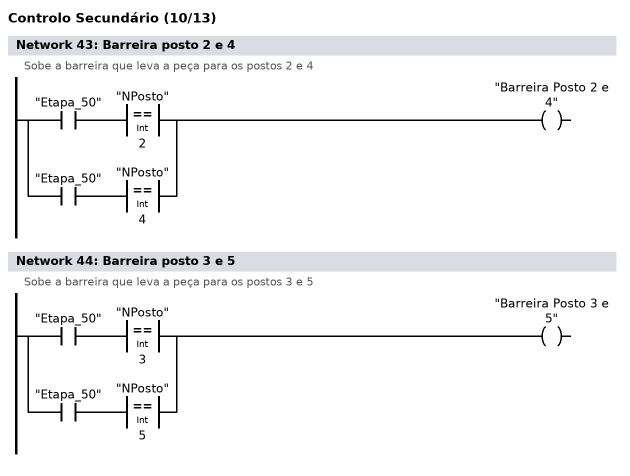
   RUNG wire#powerrail
      Contact( "Etapa_50" )
      { S7_Templates := "SrcType := Int" } EQ_Contact(in1 := "NPosto", in2 := 2)
      wire#w1
      Coil( "Barreira Posto 2 e 4" )
   END_RUNG
   RUNG wire#powerrail
      Contact( "Etapa_50" )
      { S7_Templates := "SrcType := Int" } EQ_Contact(in1 := "NPosto", in2 := 4)
   END_RUNG wire#w1
   // the same network as SCL:
   "Barreira Posto 2 e 4" := ("Etapa_50" AND ("NPosto" = 2)) OR ("Etapa_50" AND ("NPosto" = 4));
END_REGION

REGION Network 44: Barreira posto 3 e 5
   // Sobe a barreira que leva a peça para os postos 3 e 5
   RUNG wire#powerrail
      Contact( "Etapa_50" )
      { S7_Templates := "SrcType := Int" } EQ_Contact(in1 := "NPosto", in2 := 3)
      wire#w1
      Coil( "Barreira Posto 3 e 5" )
   END_RUNG
   RUNG wire#powerrail
      Contact( "Etapa_50" )
      { S7_Templates := "SrcType := Int" } EQ_Contact(in1 := "NPosto", in2 := 5)
   END_RUNG wire#w1
   // the same network as SCL:
   "Barreira Posto 3 e 5" := ("Etapa_50" AND ("NPosto" = 3)) OR ("Etapa_50" AND ("NPosto" = 5));
END_REGION

REGION Network 45: Contadores de postos
   // Incrementa os contadores dos postos de armazenamento individuais e do contador total
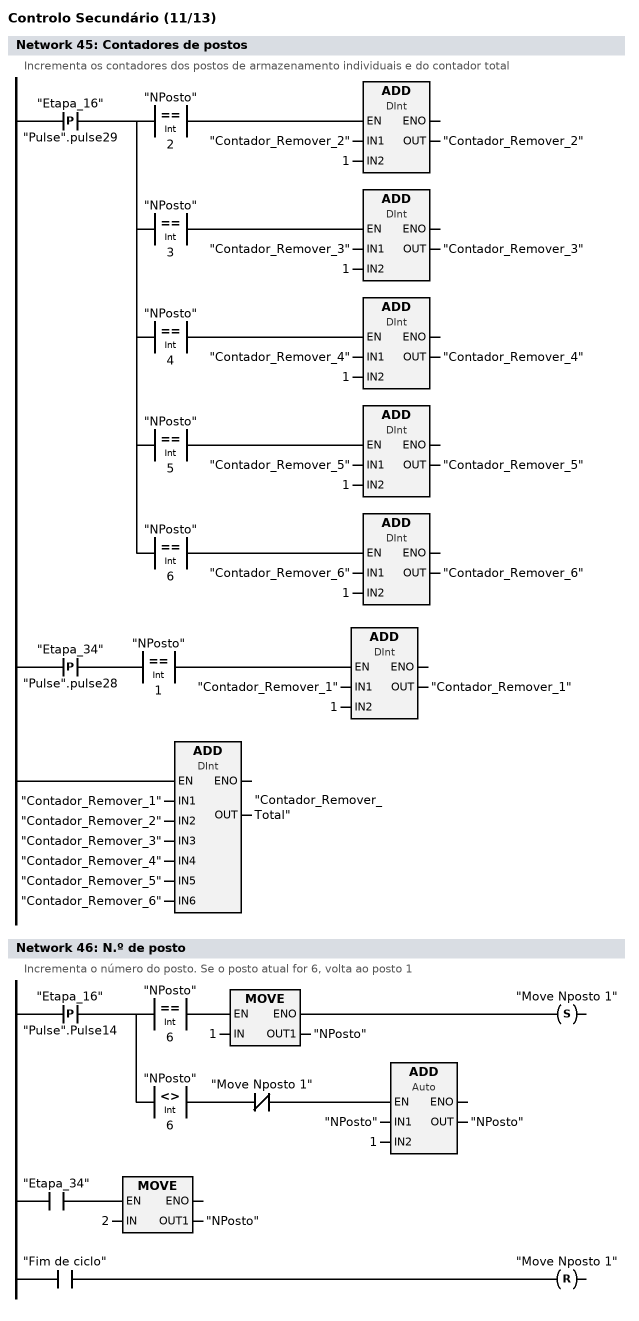
   RUNG wire#powerrail
      P_Contact(operand := "Etapa_16", bit := "Pulse".pulse29)
      wire#w1
      { S7_Templates := "SrcType := Int" } EQ_Contact(in1 := "NPosto", in2 := 2)
      { S7_Templates := "SrcType := DInt" } Add(in1 := "Contador_Remover_2", in2 := 1, out => "Contador_Remover_2")
   END_RUNG
   RUNG wire#w1
      { S7_Templates := "SrcType := Int" } EQ_Contact(in1 := "NPosto", in2 := 3)
      { S7_Templates := "SrcType := DInt" } Add(in1 := "Contador_Remover_3", in2 := 1, out => "Contador_Remover_3")
   END_RUNG
   RUNG wire#w1
      { S7_Templates := "SrcType := Int" } EQ_Contact(in1 := "NPosto", in2 := 4)
      { S7_Templates := "SrcType := DInt" } Add(in1 := "Contador_Remover_4", in2 := 1, out => "Contador_Remover_4")
   END_RUNG
   RUNG wire#w1
      { S7_Templates := "SrcType := Int" } EQ_Contact(in1 := "NPosto", in2 := 5)
      { S7_Templates := "SrcType := DInt" } Add(in1 := "Contador_Remover_5", in2 := 1, out => "Contador_Remover_5")
   END_RUNG
   RUNG wire#w1
      { S7_Templates := "SrcType := Int" } EQ_Contact(in1 := "NPosto", in2 := 6)
      { S7_Templates := "SrcType := DInt" } Add(in1 := "Contador_Remover_6", in2 := 1, out => "Contador_Remover_6")
   END_RUNG
   RUNG wire#powerrail
      P_Contact(operand := "Etapa_34", bit := "Pulse".pulse28)
      { S7_Templates := "SrcType := Int" } EQ_Contact(in1 := "NPosto", in2 := 1)
      { S7_Templates := "SrcType := DInt" } Add(in1 := "Contador_Remover_1", in2 := 1, out => "Contador_Remover_1")
   END_RUNG
   RUNG wire#powerrail
      { S7_Templates := "SrcType := DInt" } Add(in1 := "Contador_Remover_1", in2 := "Contador_Remover_2", in3 := "Contador_Remover_3", in4 := "Contador_Remover_4", in5 := "Contador_Remover_5", in6 := "Contador_Remover_6", out => "Contador_Remover_Total")
   END_RUNG
   // the same network as SCL:
   #_w1 := "Etapa_16" AND NOT "Pulse".pulse29;   // rising edge of "Etapa_16"
   "Pulse".pulse29 := "Etapa_16";
   IF #_w1 AND ("NPosto" = 2) THEN "Contador_Remover_2" := "Contador_Remover_2" + 1; END_IF;
   IF #_w1 AND ("NPosto" = 3) THEN "Contador_Remover_3" := "Contador_Remover_3" + 1; END_IF;
   IF #_w1 AND ("NPosto" = 4) THEN "Contador_Remover_4" := "Contador_Remover_4" + 1; END_IF;
   IF #_w1 AND ("NPosto" = 5) THEN "Contador_Remover_5" := "Contador_Remover_5" + 1; END_IF;
   IF #_w1 AND ("NPosto" = 6) THEN "Contador_Remover_6" := "Contador_Remover_6" + 1; END_IF;
   #_w2 := "Etapa_34" AND NOT "Pulse".pulse28;   // rising edge of "Etapa_34"
   "Pulse".pulse28 := "Etapa_34";
   IF #_w2 AND ("NPosto" = 1) THEN "Contador_Remover_1" := "Contador_Remover_1" + 1; END_IF;
   "Contador_Remover_Total" := "Contador_Remover_1" + "Contador_Remover_2" + "Contador_Remover_3" + "Contador_Remover_4" + "Contador_Remover_5" + "Contador_Remover_6";
END_REGION

REGION Network 46: N.º de posto
   // Incrementa o número do posto. Se o posto atual for 6, volta ao posto 1
   RUNG wire#powerrail
      P_Contact(operand := "Etapa_16", bit := "Pulse".Pulse14)
      wire#w1
      { S7_Templates := "SrcType := Int" } EQ_Contact(in1 := "NPosto", in2 := 6)
      Move(in := 1, out1 => "NPosto")
      S_Coil( "Move Nposto 1" )
   END_RUNG
   RUNG wire#w1
      { S7_Templates := "SrcType := Int" } NE_Contact(in1 := "NPosto", in2 := 6)
      I_Contact( "Move Nposto 1" )
      Add(in1 := "NPosto", in2 := 1, out => "NPosto")
   END_RUNG
   RUNG wire#powerrail
      Contact( "Etapa_34" )
      Move(in := 2, out1 => "NPosto")
   END_RUNG
   RUNG wire#powerrail
      Contact( "Fim de ciclo" )
      R_Coil( "Move Nposto 1" )
   END_RUNG
   // the same network as SCL:
   #_w1 := "Etapa_16" AND NOT "Pulse".Pulse14;   // rising edge of "Etapa_16"
   "Pulse".Pulse14 := "Etapa_16";
   #_w2 := #_w1 AND ("NPosto" = 6);
   IF #_w2 THEN
       "NPosto" := 1;
       "Move Nposto 1" := TRUE;
   END_IF;
   IF #_w1 AND ("NPosto" <> 6) AND NOT "Move Nposto 1" THEN "NPosto" := "NPosto" + 1; END_IF;
   IF "Etapa_34" THEN "NPosto" := 2; END_IF;
   IF "Fim de ciclo" THEN "Move Nposto 1" := FALSE; END_IF;
END_REGION

REGION Network 47: Tapete 7
   // Permite a definição da velocidade do tapete 7. Está predefinido para 5
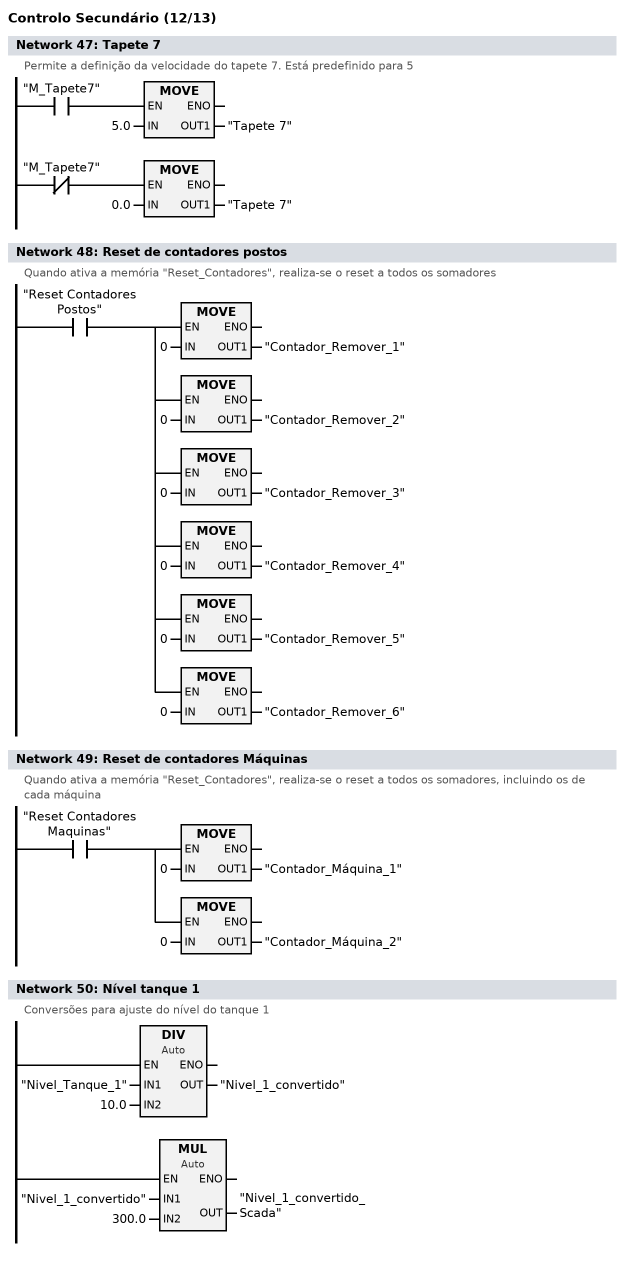
   RUNG wire#powerrail
      Contact( "M_Tapete7" )
      Move(in := 5.0, out1 => "Tapete 7")
   END_RUNG
   RUNG wire#powerrail
      I_Contact( "M_Tapete7" )
      Move(in := 0.0, out1 => "Tapete 7")
   END_RUNG
   // the same network as SCL:
   IF "M_Tapete7" THEN "Tapete 7" := 5.0; END_IF;
   IF NOT "M_Tapete7" THEN "Tapete 7" := 0.0; END_IF;
END_REGION

REGION Network 48: Reset de contadores postos
   // Quando ativa a memória "Reset_Contadores", realiza-se o reset a todos os somadores
   RUNG wire#powerrail
      Contact( "Reset Contadores Postos" )
      wire#w1
      Move(in := 0, out1 => "Contador_Remover_1")
   END_RUNG
   RUNG wire#w1
      Move(in := 0, out1 => "Contador_Remover_2")
   END_RUNG
   RUNG wire#w1
      Move(in := 0, out1 => "Contador_Remover_3")
   END_RUNG
   RUNG wire#w1
      Move(in := 0, out1 => "Contador_Remover_4")
   END_RUNG
   RUNG wire#w1
      Move(in := 0, out1 => "Contador_Remover_5")
   END_RUNG
   RUNG wire#w1
      Move(in := 0, out1 => "Contador_Remover_6")
   END_RUNG
   // the same network as SCL:
   IF "Reset Contadores Postos" THEN
       "Contador_Remover_1" := 0;
       "Contador_Remover_2" := 0;
       "Contador_Remover_3" := 0;
       "Contador_Remover_4" := 0;
       "Contador_Remover_5" := 0;
       "Contador_Remover_6" := 0;
   END_IF;
END_REGION

REGION Network 49: Reset de contadores Máquinas
   // Quando ativa a memória "Reset_Contadores", realiza-se o reset a todos os somadores, incluindo os de cada máquina
   RUNG wire#powerrail
      Contact( "Reset Contadores Maquinas" )
      wire#w1
      Move(in := 0, out1 => "Contador_Máquina_1")
   END_RUNG
   RUNG wire#w1
      Move(in := 0, out1 => "Contador_Máquina_2")
   END_RUNG
   // the same network as SCL:
   IF "Reset Contadores Maquinas" THEN
       "Contador_Máquina_1" := 0;
       "Contador_Máquina_2" := 0;
   END_IF;
END_REGION

REGION Network 50: Nível tanque 1
   // Conversões para ajuste do nível do tanque 1
   RUNG wire#powerrail
      Div(in1 := "Nivel_Tanque_1", in2 := 10.0, out => "Nivel_1_convertido")
   END_RUNG
   RUNG wire#powerrail
      Mul(in1 := "Nivel_1_convertido", in2 := 300.0, out => "Nivel_1_convertido_Scada")
   END_RUNG
   // the same network as SCL:
   "Nivel_1_convertido" := "Nivel_Tanque_1" / 10.0;
   "Nivel_1_convertido_Scada" := "Nivel_1_convertido" * 300.0;
END_REGION

REGION Network 51: Nível tanque 2
   // Conversões para ajuste do nível do tanque 2
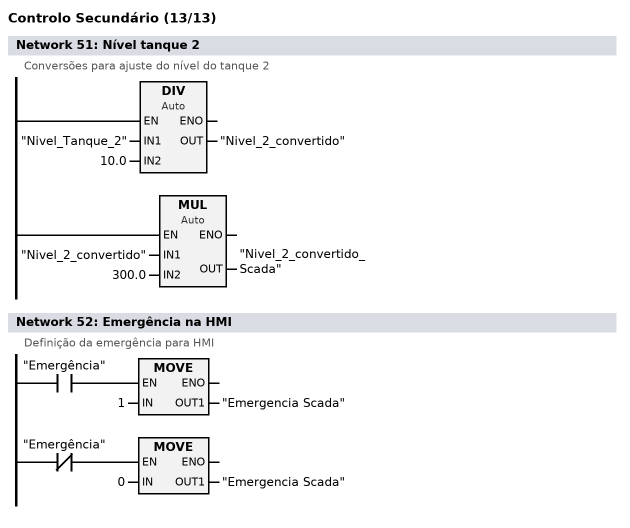
   RUNG wire#powerrail
      Div(in1 := "Nivel_Tanque_2", in2 := 10.0, out => "Nivel_2_convertido")
   END_RUNG
   RUNG wire#powerrail
      Mul(in1 := "Nivel_2_convertido", in2 := 300.0, out => "Nivel_2_convertido_Scada")
   END_RUNG
   // the same network as SCL:
   "Nivel_2_convertido" := "Nivel_Tanque_2" / 10.0;
   "Nivel_2_convertido_Scada" := "Nivel_2_convertido" * 300.0;
END_REGION

REGION Network 52: Emergência na HMI
   // Definição da emergência para HMI
   RUNG wire#powerrail
      Contact( "Emergência" )
      Move(in := 1, out1 => "Emergencia Scada")
   END_RUNG
   RUNG wire#powerrail
      I_Contact( "Emergência" )
      Move(in := 0, out1 => "Emergencia Scada")
   END_RUNG
   // the same network as SCL:
   IF "Emergência" THEN "Emergencia Scada" := 1; END_IF;
   IF NOT "Emergência" THEN "Emergencia Scada" := 0; END_IF;
END_REGION
END_FUNCTION

FUNCTION "Passadeira 3" : Void   // FC5, LAD
TITLE = Passadeira 3
{ S7_Optimized_Access := 'TRUE' }
VERSION : 0.1
   VAR_TEMP   // added for the SCL form of the ladder/FBD networks
      _w1 : Bool;
   END_VAR
BEGIN

REGION Network 1: Stop tapete 3
   // O tapete inicia ligado. Se detectar peça na saída do tapete 3, pára o tapete
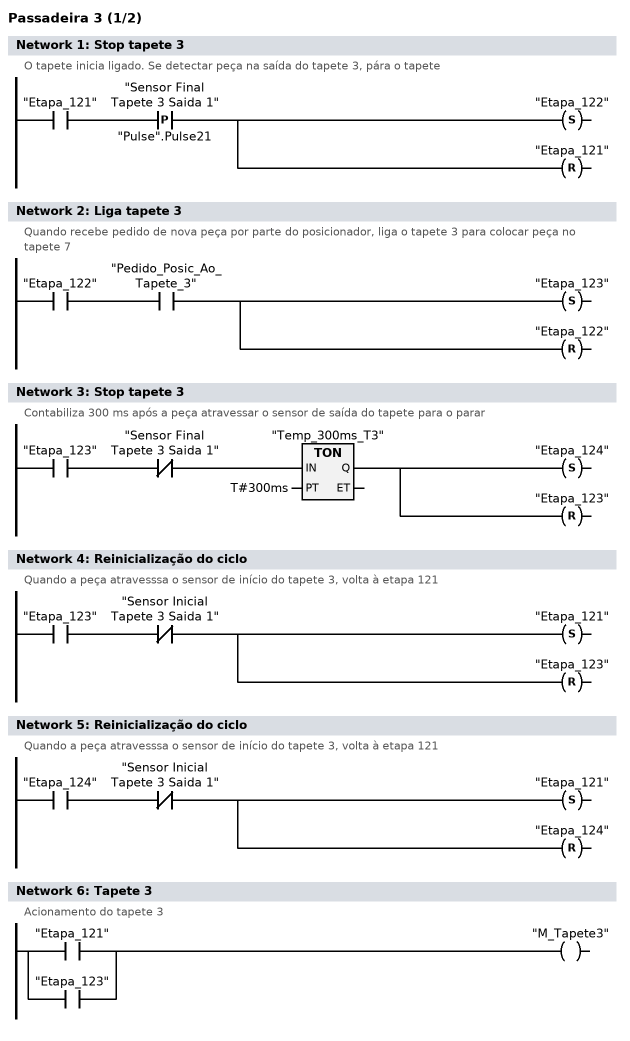
   RUNG wire#powerrail
      Contact( "Etapa_121" )
      P_Contact(operand := "Sensor Final Tapete 3 Saida 1", bit := "Pulse".Pulse21)
      wire#w1
      S_Coil( "Etapa_122" )
   END_RUNG
   RUNG wire#w1
      R_Coil( "Etapa_121" )
   END_RUNG
   // the same network as SCL:
   #_w1 := "Etapa_121" AND "Sensor Final Tapete 3 Saida 1" AND NOT "Pulse".Pulse21;   // rising edge of "Sensor Final Tapete 3 Saida 1"
   "Pulse".Pulse21 := "Sensor Final Tapete 3 Saida 1";
   IF #_w1 THEN
       "Etapa_122" := TRUE;
       "Etapa_121" := FALSE;
   END_IF;
END_REGION

REGION Network 2: Liga tapete 3
   // Quando recebe pedido de nova peça por parte do posicionador, liga o tapete 3 para colocar peça no tapete 7
   RUNG wire#powerrail
      Contact( "Etapa_122" )
      Contact( "Pedido_Posic_Ao_Tapete_3" )
      wire#w1
      S_Coil( "Etapa_123" )
   END_RUNG
   RUNG wire#w1
      R_Coil( "Etapa_122" )
   END_RUNG
   // the same network as SCL:
   IF "Etapa_122" AND "Pedido_Posic_Ao_Tapete_3" THEN
       "Etapa_123" := TRUE;
       "Etapa_122" := FALSE;
   END_IF;
END_REGION

REGION Network 3: Stop tapete 3
   // Contabiliza 300 ms após a peça atravessar o sensor de saída do tapete para o parar
   "Temp_300ms_T3".TON(IN := "Etapa_123" AND NOT "Sensor Final Tapete 3 Saida 1", PT := T#300ms);
   IF "Temp_300ms_T3".Q THEN
       "Etapa_124" := TRUE;
       "Etapa_123" := FALSE;
   END_IF;
END_REGION

REGION Network 4: Reinicialização do ciclo
   // Quando a peça atravesssa o sensor de início do tapete 3, volta à etapa 121
   RUNG wire#powerrail
      Contact( "Etapa_123" )
      I_Contact( "Sensor Inicial Tapete 3 Saida 1" )
      wire#w1
      S_Coil( "Etapa_121" )
   END_RUNG
   RUNG wire#w1
      R_Coil( "Etapa_123" )
   END_RUNG
   // the same network as SCL:
   IF "Etapa_123" AND NOT "Sensor Inicial Tapete 3 Saida 1" THEN
       "Etapa_121" := TRUE;
       "Etapa_123" := FALSE;
   END_IF;
END_REGION

REGION Network 5: Reinicialização do ciclo
   // Quando a peça atravesssa o sensor de início do tapete 3, volta à etapa 121
   RUNG wire#powerrail
      Contact( "Etapa_124" )
      I_Contact( "Sensor Inicial Tapete 3 Saida 1" )
      wire#w1
      S_Coil( "Etapa_121" )
   END_RUNG
   RUNG wire#w1
      R_Coil( "Etapa_124" )
   END_RUNG
   // the same network as SCL:
   IF "Etapa_124" AND NOT "Sensor Inicial Tapete 3 Saida 1" THEN
       "Etapa_121" := TRUE;
       "Etapa_124" := FALSE;
   END_IF;
END_REGION

REGION Network 6: Tapete 3
   // Acionamento do tapete 3
   RUNG wire#powerrail
      Contact( "Etapa_121" )
      wire#w1
      Coil( "M_Tapete3" )
   END_RUNG
   RUNG wire#powerrail
      Contact( "Etapa_123" )
   END_RUNG wire#w1
   // the same network as SCL:
   "M_Tapete3" := "Etapa_121" OR "Etapa_123";
END_REGION

REGION Network 7: Velocidade tapete 3
   // Permite a definição da velocidade do tapete 3. Está predefinido para 5
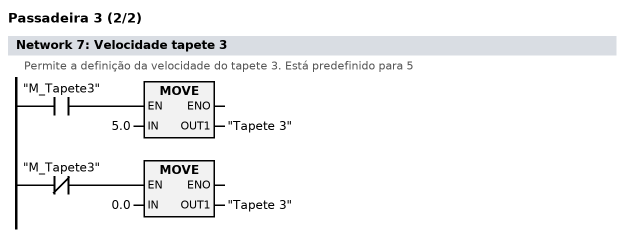
   RUNG wire#powerrail
      Contact( "M_Tapete3" )
      Move(in := 5.0, out1 => "Tapete 3")
   END_RUNG
   RUNG wire#powerrail
      I_Contact( "M_Tapete3" )
      Move(in := 0.0, out1 => "Tapete 3")
   END_RUNG
   // the same network as SCL:
   IF "M_Tapete3" THEN "Tapete 3" := 5.0; END_IF;
   IF NOT "M_Tapete3" THEN "Tapete 3" := 0.0; END_IF;
END_REGION
END_FUNCTION

FUNCTION "Passadeira 4" : Void   // FC6, LAD
TITLE = Passadeira 4
{ S7_Optimized_Access := 'TRUE' }
VERSION : 0.1
   VAR_TEMP   // added for the SCL form of the ladder/FBD networks
      _w1 : Bool;
   END_VAR
BEGIN

REGION Network 1: Stop tapete 4
   // O tapete inicia ligado. Se detectar peça na saída do tapete 4, pára o tapete
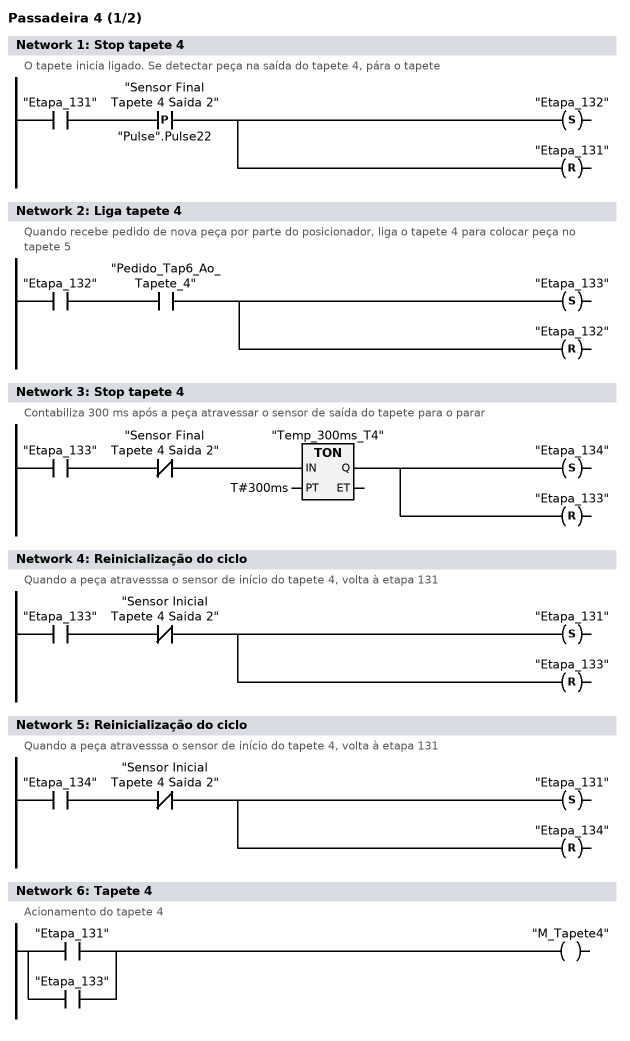
   RUNG wire#powerrail
      Contact( "Etapa_131" )
      P_Contact(operand := "Sensor Final Tapete 4 Saida 2", bit := "Pulse".Pulse22)
      wire#w1
      S_Coil( "Etapa_132" )
   END_RUNG
   RUNG wire#w1
      R_Coil( "Etapa_131" )
   END_RUNG
   // the same network as SCL:
   #_w1 := "Etapa_131" AND "Sensor Final Tapete 4 Saida 2" AND NOT "Pulse".Pulse22;   // rising edge of "Sensor Final Tapete 4 Saida 2"
   "Pulse".Pulse22 := "Sensor Final Tapete 4 Saida 2";
   IF #_w1 THEN
       "Etapa_132" := TRUE;
       "Etapa_131" := FALSE;
   END_IF;
END_REGION

REGION Network 2: Liga tapete 4
   // Quando recebe pedido de nova peça por parte do posicionador, liga o tapete 4 para colocar peça no tapete 5
   RUNG wire#powerrail
      Contact( "Etapa_132" )
      Contact( "Pedido_Tap6_Ao_Tapete_4" )
      wire#w1
      S_Coil( "Etapa_133" )
   END_RUNG
   RUNG wire#w1
      R_Coil( "Etapa_132" )
   END_RUNG
   // the same network as SCL:
   IF "Etapa_132" AND "Pedido_Tap6_Ao_Tapete_4" THEN
       "Etapa_133" := TRUE;
       "Etapa_132" := FALSE;
   END_IF;
END_REGION

REGION Network 3: Stop tapete 4
   // Contabiliza 300 ms após a peça atravessar o sensor de saída do tapete para o parar
   "Temp_300ms_T4".TON(IN := "Etapa_133" AND NOT "Sensor Final Tapete 4 Saida 2", PT := T#300ms);
   IF "Temp_300ms_T4".Q THEN
       "Etapa_134" := TRUE;
       "Etapa_133" := FALSE;
   END_IF;
END_REGION

REGION Network 4: Reinicialização do ciclo
   // Quando a peça atravesssa o sensor de início do tapete 4, volta à etapa 131
   RUNG wire#powerrail
      Contact( "Etapa_133" )
      I_Contact( "Sensor Inicial Tapete 4 Saida 2" )
      wire#w1
      S_Coil( "Etapa_131" )
   END_RUNG
   RUNG wire#w1
      R_Coil( "Etapa_133" )
   END_RUNG
   // the same network as SCL:
   IF "Etapa_133" AND NOT "Sensor Inicial Tapete 4 Saida 2" THEN
       "Etapa_131" := TRUE;
       "Etapa_133" := FALSE;
   END_IF;
END_REGION

REGION Network 5: Reinicialização do ciclo
   // Quando a peça atravesssa o sensor de início do tapete 4, volta à etapa 131
   RUNG wire#powerrail
      Contact( "Etapa_134" )
      I_Contact( "Sensor Inicial Tapete 4 Saida 2" )
      wire#w1
      S_Coil( "Etapa_131" )
   END_RUNG
   RUNG wire#w1
      R_Coil( "Etapa_134" )
   END_RUNG
   // the same network as SCL:
   IF "Etapa_134" AND NOT "Sensor Inicial Tapete 4 Saida 2" THEN
       "Etapa_131" := TRUE;
       "Etapa_134" := FALSE;
   END_IF;
END_REGION

REGION Network 6: Tapete 4
   // Acionamento do tapete 4
   RUNG wire#powerrail
      Contact( "Etapa_131" )
      wire#w1
      Coil( "M_Tapete4" )
   END_RUNG
   RUNG wire#powerrail
      Contact( "Etapa_133" )
   END_RUNG wire#w1
   // the same network as SCL:
   "M_Tapete4" := "Etapa_131" OR "Etapa_133";
END_REGION

REGION Network 7: Velocidade tapete 4
   // Permite a definição da velocidade do tapete 4. Está predefinido para 5
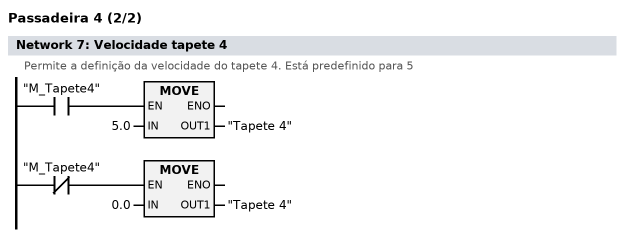
   RUNG wire#powerrail
      Contact( "M_Tapete4" )
      Move(in := 5.0, out1 => "Tapete 4")
   END_RUNG
   RUNG wire#powerrail
      I_Contact( "M_Tapete4" )
      Move(in := 0.0, out1 => "Tapete 4")
   END_RUNG
   // the same network as SCL:
   IF "M_Tapete4" THEN "Tapete 4" := 5.0; END_IF;
   IF NOT "M_Tapete4" THEN "Tapete 4" := 0.0; END_IF;
END_REGION
END_FUNCTION

FUNCTION "Passadeira 5 e 6" : Void   // FC7, LAD
TITLE = Passadeira 5 e 6
{ S7_Optimized_Access := 'TRUE' }
VERSION : 0.1
   VAR_TEMP   // added for the SCL form of the ladder/FBD networks
      _w1 : Bool;
   END_VAR
BEGIN

REGION Network 1: Stop tapete 5 e 6
   // Os tapetes 5 e 6 iniciam ligados e permanecem durante 3s para verificar se tem alguma peça a meio do tapete. Se durante 3s não detetar peça no final do tapete 6, pára os dois tapetes
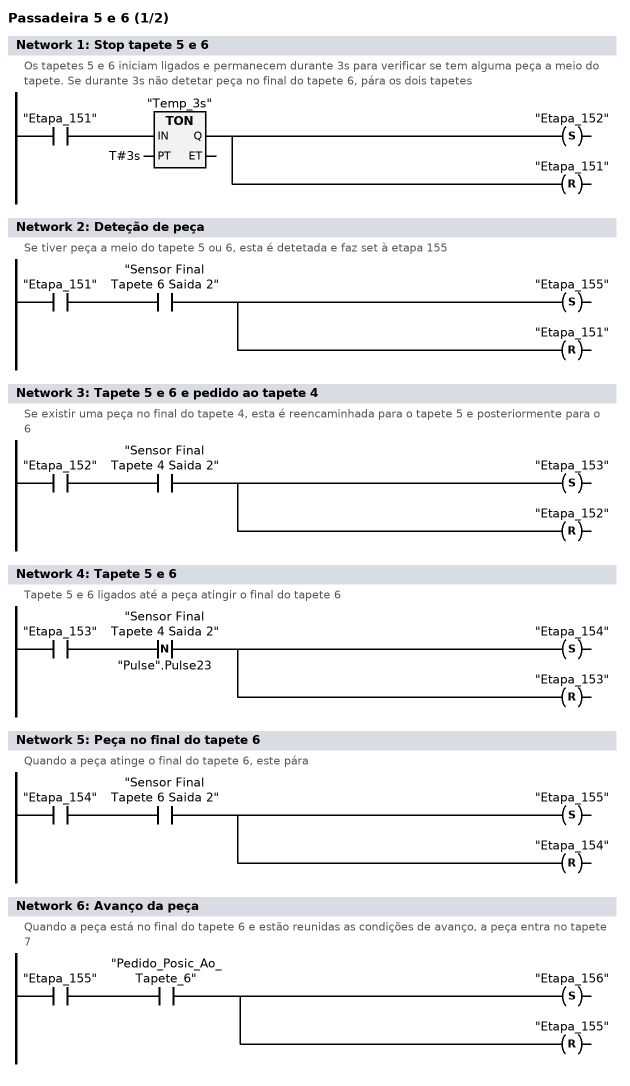
   "Temp_3s".TON(IN := "Etapa_151", PT := T#3s);
   IF "Temp_3s".Q THEN
       "Etapa_152" := TRUE;
       "Etapa_151" := FALSE;
   END_IF;
END_REGION

REGION Network 2: Deteção de peça
   // Se tiver peça a meio do tapete 5 ou 6, esta é detetada e faz set à etapa 155
   RUNG wire#powerrail
      Contact( "Etapa_151" )
      Contact( "Sensor Final Tapete 6 Saida 2" )
      wire#w1
      S_Coil( "Etapa_155" )
   END_RUNG
   RUNG wire#w1
      R_Coil( "Etapa_151" )
   END_RUNG
   // the same network as SCL:
   IF "Etapa_151" AND "Sensor Final Tapete 6 Saida 2" THEN
       "Etapa_155" := TRUE;
       "Etapa_151" := FALSE;
   END_IF;
END_REGION

REGION Network 3: Tapete 5 e 6 e pedido ao tapete 4
   // Se existir uma peça no final do tapete 4, esta é reencaminhada para o tapete 5 e posteriormente para o 6
   RUNG wire#powerrail
      Contact( "Etapa_152" )
      Contact( "Sensor Final Tapete 4 Saida 2" )
      wire#w1
      S_Coil( "Etapa_153" )
   END_RUNG
   RUNG wire#w1
      R_Coil( "Etapa_152" )
   END_RUNG
   // the same network as SCL:
   IF "Etapa_152" AND "Sensor Final Tapete 4 Saida 2" THEN
       "Etapa_153" := TRUE;
       "Etapa_152" := FALSE;
   END_IF;
END_REGION

REGION Network 4: Tapete 5 e 6
   // Tapete 5 e 6 ligados até a peça atingir o final do tapete 6
   RUNG wire#powerrail
      Contact( "Etapa_153" )
      N_Contact(operand := "Sensor Final Tapete 4 Saida 2", bit := "Pulse".Pulse23)
      wire#w1
      S_Coil( "Etapa_154" )
   END_RUNG
   RUNG wire#w1
      R_Coil( "Etapa_153" )
   END_RUNG
   // the same network as SCL:
   #_w1 := "Etapa_153" AND NOT "Sensor Final Tapete 4 Saida 2" AND "Pulse".Pulse23;   // falling edge of "Sensor Final Tapete 4 Saida 2"
   "Pulse".Pulse23 := "Sensor Final Tapete 4 Saida 2";
   IF #_w1 THEN
       "Etapa_154" := TRUE;
       "Etapa_153" := FALSE;
   END_IF;
END_REGION

REGION Network 5: Peça no final do tapete 6
   // Quando a peça atinge o final do tapete 6, este pára
   RUNG wire#powerrail
      Contact( "Etapa_154" )
      Contact( "Sensor Final Tapete 6 Saida 2" )
      wire#w1
      S_Coil( "Etapa_155" )
   END_RUNG
   RUNG wire#w1
      R_Coil( "Etapa_154" )
   END_RUNG
   // the same network as SCL:
   IF "Etapa_154" AND "Sensor Final Tapete 6 Saida 2" THEN
       "Etapa_155" := TRUE;
       "Etapa_154" := FALSE;
   END_IF;
END_REGION

REGION Network 6: Avanço da peça
   // Quando a peça está no final do tapete 6 e estão reunidas as condições de avanço, a peça entra no tapete 7
   RUNG wire#powerrail
      Contact( "Etapa_155" )
      Contact( "Pedido_Posic_Ao_Tapete_6" )
      wire#w1
      S_Coil( "Etapa_156" )
   END_RUNG
   RUNG wire#w1
      R_Coil( "Etapa_155" )
   END_RUNG
   // the same network as SCL:
   IF "Etapa_155" AND "Pedido_Posic_Ao_Tapete_6" THEN
       "Etapa_156" := TRUE;
       "Etapa_155" := FALSE;
   END_IF;
END_REGION

REGION Network 7: Fim de ciclo
   // Quando a peça sai do tapete 6, espera 300ms e faz-se set à etapa 152
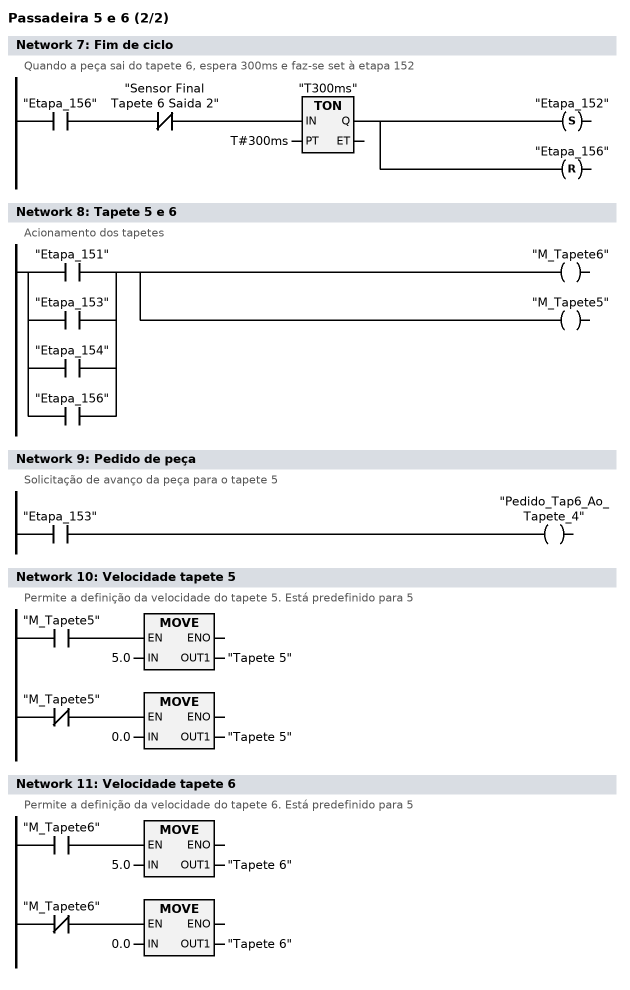
   "T300ms".TON(IN := "Etapa_156" AND NOT "Sensor Final Tapete 6 Saida 2", PT := T#300ms);
   IF "T300ms".Q THEN
       "Etapa_152" := TRUE;
       "Etapa_156" := FALSE;
   END_IF;
END_REGION

REGION Network 8: Tapete 5 e 6
   // Acionamento dos tapetes
   RUNG wire#powerrail
      Contact( "Etapa_151" )
      wire#w1
      Coil( "M_Tapete6" )
   END_RUNG
   RUNG wire#powerrail
      Contact( "Etapa_153" )
   END_RUNG wire#w1
   RUNG wire#powerrail
      Contact( "Etapa_154" )
   END_RUNG wire#w1
   RUNG wire#powerrail
      Contact( "Etapa_156" )
   END_RUNG wire#w1
   RUNG wire#w1
      Coil( "M_Tapete5" )
   END_RUNG
   // the same network as SCL:
   "M_Tapete6" := "Etapa_151" OR "Etapa_153" OR "Etapa_154" OR "Etapa_156";
   "M_Tapete5" := "M_Tapete6";
END_REGION

REGION Network 9: Pedido de peça
   // Solicitação de avanço da peça para o tapete 5
   RUNG wire#powerrail
      Contact( "Etapa_153" )
      Coil( "Pedido_Tap6_Ao_Tapete_4" )
   END_RUNG
   // the same network as SCL:
   "Pedido_Tap6_Ao_Tapete_4" := "Etapa_153";
END_REGION

REGION Network 10: Velocidade tapete 5
   // Permite a definição da velocidade do tapete 5. Está predefinido para 5
   RUNG wire#powerrail
      Contact( "M_Tapete5" )
      Move(in := 5.0, out1 => "Tapete 5")
   END_RUNG
   RUNG wire#powerrail
      I_Contact( "M_Tapete5" )
      Move(in := 0.0, out1 => "Tapete 5")
   END_RUNG
   // the same network as SCL:
   IF "M_Tapete5" THEN "Tapete 5" := 5.0; END_IF;
   IF NOT "M_Tapete5" THEN "Tapete 5" := 0.0; END_IF;
END_REGION

REGION Network 11: Velocidade tapete 6
   // Permite a definição da velocidade do tapete 6. Está predefinido para 5
   RUNG wire#powerrail
      Contact( "M_Tapete6" )
      Move(in := 5.0, out1 => "Tapete 6")
   END_RUNG
   RUNG wire#powerrail
      I_Contact( "M_Tapete6" )
      Move(in := 0.0, out1 => "Tapete 6")
   END_RUNG
   // the same network as SCL:
   IF "M_Tapete6" THEN "Tapete 6" := 5.0; END_IF;
   IF NOT "M_Tapete6" THEN "Tapete 6" := 0.0; END_IF;
END_REGION
END_FUNCTION

FUNCTION "Avisos" : Void   // FC8, LAD
TITLE = Avisos
{ S7_Optimized_Access := 'TRUE' }
VERSION : 0.1
BEGIN

REGION Network 1: Aviso de nenhum posto de armazenamento habilitado na HMI
   // Quando se carrega no start e não está nenhum posto habilitado, liga um aviso durante 5 segundos na HMI
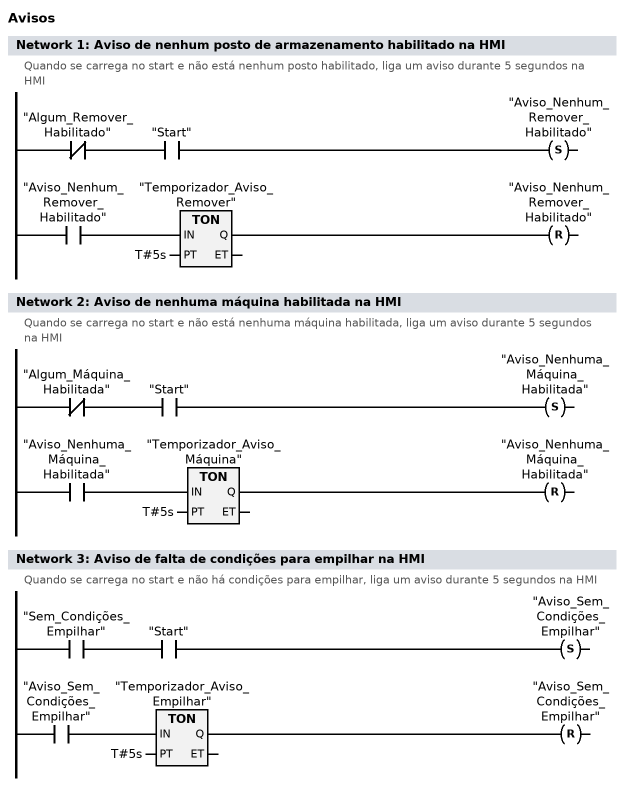
   IF NOT "Algum_Remover_Habilitado" AND "Start" THEN "Aviso_Nenhum_Remover_Habilitado" := TRUE; END_IF;
   "Temporizador_Aviso_Remover".TON(IN := "Aviso_Nenhum_Remover_Habilitado", PT := T#5s);
   IF "Temporizador_Aviso_Remover".Q THEN "Aviso_Nenhum_Remover_Habilitado" := FALSE; END_IF;
END_REGION

REGION Network 2: Aviso de nenhuma máquina habilitada na HMI
   // Quando se carrega no start e não está nenhuma máquina habilitada, liga um aviso durante 5 segundos na HMI
   IF NOT "Algum_Máquina_Habilitada" AND "Start" THEN "Aviso_Nenhuma_Máquina_Habilitada" := TRUE; END_IF;
   "Temporizador_Aviso_Máquina".TON(IN := "Aviso_Nenhuma_Máquina_Habilitada", PT := T#5s);
   IF "Temporizador_Aviso_Máquina".Q THEN "Aviso_Nenhuma_Máquina_Habilitada" := FALSE; END_IF;
END_REGION

REGION Network 3: Aviso de falta de condições para empilhar na HMI
   // Quando se carrega no start e não há condições para empilhar, liga um aviso durante 5 segundos na HMI
   IF "Sem_Condições_Empilhar" AND "Start" THEN "Aviso_Sem_Condições_Empilhar" := TRUE; END_IF;
   "Temporizador_Aviso_Empilhar".TON(IN := "Aviso_Sem_Condições_Empilhar", PT := T#5s);
   IF "Temporizador_Aviso_Empilhar".Q THEN "Aviso_Sem_Condições_Empilhar" := FALSE; END_IF;
END_REGION
END_FUNCTION

FUNCTION "Tempo_FC" : Void   // FC9, LAD
TITLE = Tempo de sistema
{ S7_Optimized_Access := 'TRUE' }
VERSION : 0.1
   VAR_TEMP   // added for the SCL form of the ladder/FBD networks
      _w1 : Bool;
   END_VAR
BEGIN

REGION Network 1: Tempo do sistema
   // Obtém a data e hora que consta no sistema
